KUKA KRL program: EPS_2_26115_SA7004_A_20260219035541.src

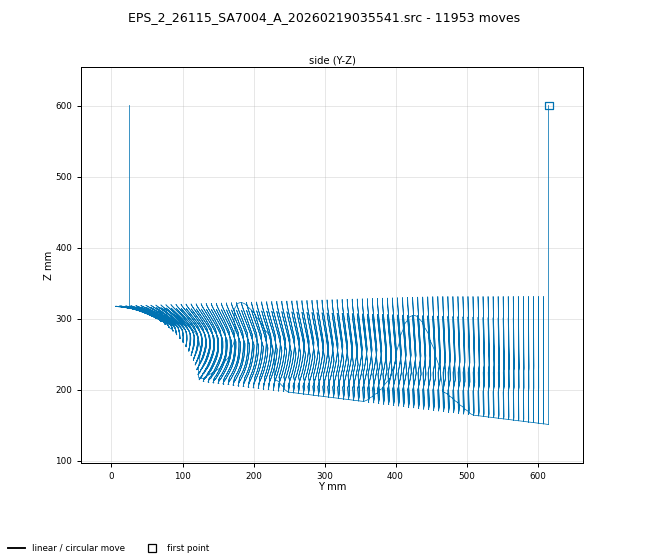
[picture p0: tool path of EPS_2_26115_SA7004_A_20260219035541.src, 11953 of 11955 moves have a stored position in this frame; points joined in program order, loops and branches not executed]
&ACCESS RVP
&REL 4
&COMMENT QRS 19112012
&PARAM EDITMASK = *
DEF PART()
EXT BAS (BAS_COMMAND :IN,REAL :IN )
INT I
BAS (#INITMOV,0 )

;KUKA QRS Post kuka4.cps  Date:22-06-2017 !

File_ID=3058

QRS_PRE_INIT()

;Init var - Until changes are made in qrs_pre_init
Outlet_Square_prg=0
Inlet_1_Square_prg=0
Inlet_2_Square_prg=0
Inlet_3_Square_prg=0
Inlet_4_Square_prg=0
Inlet_5_Square_prg=0

Outlet_1={X 0.000, Y 460.000, Z 230.500, B 0.000, E1 0.000 }
Inlet_1={X 0.000, Y 539.550, Z 200.500, B 0.000, E1 180.000 }
Outlet_1_type=201
Inlet_1_type=201
;QRS#1=Sidecore dimensions
;QRS#2=200-8" PVC SDR 35 Cut Back
;QRS#3=200-8" PVC SDR 35
;QRS#4=
;QRS#5=
;QRS#6=
;QRS#7=
;QRS#8=
;QRS#9=12-08 PSX
;QRS#10=12-08 PSX
;QRS#11=
;QRS#12=
;QRS#13=
;QRS#14=
;QRS#15=
;QRS#16=1220x127x610 2'
;QRS#17=EPS Height
;QRS#18=331
;QRS#19=*
;QRS#20= UPDATED VERSION 22-06-2017
;QRS#21=*
Outlet_Square=0100
Inlet_1_Square=0100
Inlet_2_Square=0
Inlet_3_Square=0
Inlet_4_Square=0
Inlet_5_Square=0
Mill_Square=1
Outlet_Square_Prg=214
Inlet_1_Square_prg=204

QRS_INIT()

$ADVANCE=5

; T1
PTP {E1 173.62,E2 173.62}
PTP {X 0,Y 615.488,A -85,B 0,C 180,E1 173.62,E2 173.62,E3 0,E4 0,E5 0,E6 0}
QRS_SPEED_INIT()
LIN {X 0,Y 615.488,Z 600,A -85,B 0,C 180,E1 173.62,E2 173.62,E3 0,E4 0,E5 0,E6 0} C_VEL
LIN {X 0,Y 615.488,Z 160.871,A -85,B 0,C 180,E1 173.62,E2 173.62} C_VEL
LIN {X 0,Y 615.488,Z 152.699,A -85,B 0,C 180,E1 173.62,E2 173.62} C_VEL
LIN {X 0,Y 615.469,Z 150.699,A -85,B 0,C 180,E1 173.434,E2 173.434} C_VEL
LIN {X 0,Y 615.452,Z 150.696,A -85,B 0,C 180,E1 170.801,E2 170.801} C_VEL
LIN {X 0,Y 615.484,Z 150.7,A -85,B 0,C 180,E1 168.139,E2 168.139} C_VEL
LIN {X 0,Y 615.492,Z 150.686,A -85,B 0,C 180,E1 165.451,E2 165.451} C_VEL
LIN {X 0,Y 615.483,Z 150.699,A -85,B 0,C 180,E1 162.729,E2 162.729} C_VEL
LIN {X 0,Y 615.468,Z 150.694,A -85,B 0,C 180,E1 159.966,E2 159.966} C_VEL
LIN {X 0,Y 615.439,Z 150.7,A -85,B 0,C 180,E1 157.153,E2 157.153} C_VEL
LIN {X 0,Y 615.449,Z 150.697,A -85,B 0,C 180,E1 155.006,E2 155.006} C_VEL
LIN {X 0,Y 615.477,Z 150.698,A -85,B 0,C 180,E1 152.822,E2 152.822} C_VEL
LIN {X 0,Y 615.49,Z 150.688,A -85,B 0,C 180,E1 149.84,E2 149.84} C_VEL
LIN {X 0,Y 615.492,Z 150.699,A -85,B 0,C 180,E1 147.543,E2 147.543} C_VEL
LIN {X 0,Y 615.448,Z 150.698,A -85,B 0,C 180,E1 145.182,E2 145.182} C_VEL
LIN {X 0,Y 615.449,Z 150.7,A -85,B 0,C 180,E1 142.755,E2 142.755} C_VEL
LIN {X 0,Y 615.461,Z 150.694,A -85,B 0,C 180,E1 139.913,E2 139.913} C_VEL
LIN {X 0,Y 615.468,Z 150.695,A -85,B 0,C 180,E1 137.645,E2 137.645} C_VEL
LIN {X 0,Y 615.479,Z 150.691,A -85,B 0,C 180,E1 134.93,E2 134.93} C_VEL
LIN {X 0,Y 615.494,Z 150.7,A -85,B 0,C 180,E1 132.08,E2 132.08} C_VEL
LIN {X 0,Y 615.444,Z 150.699,A -85,B 0,C 180,E1 129.753,E2 129.753} C_VEL
LIN {X 0,Y 615.479,Z 150.704,A -85,B 0,C 180,E1 126.935,E2 126.935} C_VEL
LIN {X 0,Y 615.451,Z 150.699,A -85,B 0,C 180,E1 125.618,E2 125.618} C_VEL
LIN {X 0,Y 615.483,Z 151.858,A -85,B 0,C 180,E1 124.7,E2 124.7} C_VEL
LIN {X 0,Y 615.454,Z 156.021,A -85,B 0,C 180,E1 122.325,E2 122.325} C_VEL
LIN {X 0,Y 615.48,Z 160.511,A -85,B 0,C 180,E1 119.793,E2 119.793} C_VEL
LIN {X 0,Y 615.495,Z 165.513,A -85,B 0,C 180,E1 117.046,E2 117.046} C_VEL
LIN {X 0,Y 615.487,Z 170.773,A -85,B 0,C 180,E1 114.272,E2 114.272} C_VEL
LIN {X 0,Y 615.488,Z 176.264,A -85,B 0,C 180,E1 111.432,E2 111.432} C_VEL
LIN {X 0,Y 615.49,Z 181.84,A -85,B 0,C 180,E1 108.605,E2 108.605} C_VEL
LIN {X 0,Y 615.465,Z 187.255,A -85,B 0,C 180,E1 105.906,E2 105.906} C_VEL
LIN {X 0,Y 615.495,Z 192.741,A -85,B 0,C 180,E1 103.201,E2 103.201} C_VEL
LIN {X 0,Y 615.492,Z 196.091,A -85,B 0,C 180,E1 101.568,E2 101.568} C_VEL
LIN {X 0,Y 615.483,Z 210.748,A -85,B 0,C 180,E1 101.235,E2 101.235} C_VEL
LIN {X 0,Y 615.446,Z 223.1,A -85,B 0,C 180,E1 100.825,E2 100.825} C_VEL
LIN {X 0,Y 615.441,Z 235.207,A -85,B 0,C 180,E1 100.278,E2 100.278} C_VEL
LIN {X 0,Y 615.493,Z 246.579,A -85,B 0,C 180,E1 99.613,E2 99.613} C_VEL
LIN {X 0,Y 615.498,Z 256.825,A -85,B 0,C 180,E1 98.867,E2 98.867} C_VEL
LIN {X 0,Y 615.498,Z 266.036,A -85,B 0,C 180,E1 98.04,E2 98.04} C_VEL
LIN {X 0,Y 615.499,Z 274.893,A -85,B 0,C 180,E1 97.057,E2 97.057} C_VEL
LIN {X 0,Y 615.497,Z 282.125,A -85,B 0,C 180,E1 96.063,E2 96.063} C_VEL
LIN {X 0,Y 615.497,Z 286.959,A -85,B 0,C 180,E1 95.241,E2 95.241} C_VEL
LIN {X 0,Y 615.494,Z 291.659,A -85,B 0,C 180,E1 94.256,E2 94.256} C_VEL
LIN {X 0,Y 615.494,Z 295.255,A -85,B 0,C 180,E1 93.273,E2 93.273} C_VEL
LIN {X 0,Y 615.496,Z 297.115,A -85,B 0,C 180,E1 92.618,E2 92.618} C_VEL
LIN {X 0,Y 615.5,Z 298.533,A -85,B 0,C 180,E1 91.963,E2 91.963} C_VEL
LIN {X 0,Y 615.496,Z 300.142,A -85,B 0,C 180,E1 90.654,E2 90.654} C_VEL
LIN {X 0,Y 615.495,Z 300.384,A -85,B 0,C 180,E1 90,E2 90} C_VEL
LIN {X 0,Y 615.495,Z 300.205,A -85,B 0,C 180,E1 89.346,E2 89.346} C_VEL
LIN {X 0,Y 615.499,Z 298.682,A -85,B 0,C 180,E1 88.037,E2 88.037} C_VEL
LIN {X 0,Y 615.498,Z 297.341,A -85,B 0,C 180,E1 87.382,E2 87.382} C_VEL
LIN {X 0,Y 615.496,Z 294.494,A -85,B 0,C 180,E1 86.399,E2 86.399} C_VEL
LIN {X 0,Y 615.498,Z 290.634,A -85,B 0,C 180,E1 85.415,E2 85.415} C_VEL
LIN {X 0,Y 615.498,Z 285.651,A -85,B 0,C 180,E1 84.43,E2 84.43} C_VEL
LIN {X 0,Y 615.496,Z 279.208,A -85,B 0,C 180,E1 83.418,E2 83.418} C_VEL
LIN {X 0,Y 615.497,Z 271.535,A -85,B 0,C 180,E1 82.454,E2 82.454} C_VEL
LIN {X 0,Y 615.498,Z 261.757,A -85,B 0,C 180,E1 81.463,E2 81.463} C_VEL
LIN {X 0,Y 615.498,Z 251.491,A -85,B 0,C 180,E1 80.636,E2 80.636} C_VEL
LIN {X 0,Y 615.447,Z 239.935,A -85,B 0,C 180,E1 79.888,E2 79.888} C_VEL
LIN {X 0,Y 615.431,Z 228.385,A -85,B 0,C 180,E1 79.305,E2 79.305} C_VEL
LIN {X 0,Y 615.463,Z 216.445,A -85,B 0,C 180,E1 78.848,E2 78.848} C_VEL
LIN {X 0,Y 615.49,Z 204.378,A -85,B 0,C 180,E1 78.515,E2 78.515} C_VEL
LIN {X 0,Y 615.489,Z 196.104,A -85,B 0,C 180,E1 78.348,E2 78.348} C_VEL
LIN {X 0,Y 615.458,Z 191.469,A -85,B 0,C 180,E1 76.08,E2 76.08} C_VEL
LIN {X 0,Y 615.458,Z 186.396,A -85,B 0,C 180,E1 73.579,E2 73.579} C_VEL
LIN {X 0,Y 615.487,Z 180.568,A -85,B 0,C 180,E1 70.662,E2 70.662} C_VEL
LIN {X 0,Y 615.477,Z 175.065,A -85,B 0,C 180,E1 67.863,E2 67.863} C_VEL
LIN {X 0,Y 615.488,Z 169.567,A -85,B 0,C 180,E1 65.008,E2 65.008} C_VEL
LIN {X 0,Y 615.484,Z 164.066,A -85,B 0,C 180,E1 62.085,E2 62.085} C_VEL
LIN {X 0,Y 615.466,Z 160.02,A -85,B 0,C 180,E1 59.839,E2 59.839} C_VEL
LIN {X 0,Y 615.462,Z 155.943,A -85,B 0,C 180,E1 57.541,E2 57.541} C_VEL
LIN {X 0,Y 615.495,Z 151.812,A -85,B 0,C 180,E1 55.185,E2 55.185} C_VEL
LIN {X 0,Y 615.464,Z 150.698,A -85,B 0,C 180,E1 54.383,E2 54.383} C_VEL
LIN {X 0,Y 615.437,Z 150.7,A -85,B 0,C 180,E1 51.928,E2 51.928} C_VEL
LIN {X 0,Y 615.49,Z 150.696,A -85,B 0,C 180,E1 49.394,E2 49.394} C_VEL
LIN {X 0,Y 615.463,Z 150.694,A -85,B 0,C 180,E1 46.753,E2 46.753} C_VEL
LIN {X 0,Y 615.481,Z 150.692,A -85,B 0,C 180,E1 43.997,E2 43.997} C_VEL
LIN {X 0,Y 615.491,Z 150.7,A -85,B 0,C 180,E1 41.095,E2 41.095} C_VEL
LIN {X 0,Y 615.453,Z 150.7,A -85,B 0,C 180,E1 38.907,E2 38.907} C_VEL
LIN {X 0,Y 615.441,Z 150.7,A -85,B 0,C 180,E1 36.428,E2 36.428} C_VEL
LIN {X 0,Y 615.467,Z 150.693,A -85,B 0,C 180,E1 33.531,E2 33.531} C_VEL
LIN {X 0,Y 615.485,Z 150.698,A -85,B 0,C 180,E1 30.92,E2 30.92} C_VEL
LIN {X 0,Y 615.479,Z 150.691,A -85,B 0,C 180,E1 28.449,E2 28.449} C_VEL
LIN {X 0,Y 615.493,Z 150.7,A -85,B 0,C 180,E1 25.57,E2 25.57} C_VEL
LIN {X 0,Y 615.458,Z 150.7,A -85,B 0,C 180,E1 23.558,E2 23.558} C_VEL
LIN {X 0,Y 615.432,Z 150.7,A -85,B 0,C 180,E1 21.434,E2 21.434} C_VEL
LIN {X 0,Y 615.494,Z 150.696,A -85,B 0,C 180,E1 18.606,E2 18.606} C_VEL
LIN {X 0,Y 615.472,Z 150.693,A -85,B 0,C 180,E1 15.906,E2 15.906} C_VEL
LIN {X 0,Y 615.475,Z 150.694,A -85,B 0,C 180,E1 13.202,E2 13.202} C_VEL
LIN {X 0,Y 615.492,Z 150.693,A -85,B 0,C 180,E1 10.527,E2 10.527} C_VEL
LIN {X 0,Y 615.437,Z 150.7,A -85,B 0,C 180,E1 7.876,E2 7.876} C_VEL
LIN {X 0,Y 615.474,Z 150.701,A -85,B 0,C 180,E1 5.241,E2 5.241} C_VEL
LIN {X 0,Y 615.474,Z 150.691,A -85,B 0,C 180,E1 2.618,E2 2.618} C_VEL
LIN {X 0,Y 615.487,Z 150.701,A -85,B 0,C 180,E1 0,E2 0} C_VEL
LIN {X 0,Y 615.478,Z 150.69,A -85,B 0,C 180,E1 -2.618,E2 -2.618} C_VEL
LIN {X 0,Y 615.489,Z 150.701,A -85,B 0,C 180,E1 -5.241,E2 -5.241} C_VEL
LIN {X 0,Y 615.433,Z 150.7,A -85,B 0,C 180,E1 -7.876,E2 -7.876} C_VEL
LIN {X 0,Y 615.494,Z 150.695,A -85,B 0,C 180,E1 -10.527,E2 -10.527} C_VEL
LIN {X 0,Y 615.468,Z 150.694,A -85,B 0,C 180,E1 -13.202,E2 -13.202} C_VEL
LIN {X 0,Y 615.478,Z 150.693,A -85,B 0,C 180,E1 -15.905,E2 -15.905} C_VEL
LIN {X 0,Y 615.494,Z 150.694,A -85,B 0,C 180,E1 -18.646,E2 -18.646} C_VEL
LIN {X 0,Y 615.436,Z 150.699,A -85,B 0,C 180,E1 -21.434,E2 -21.434} C_VEL
LIN {X 0,Y 615.484,Z 150.696,A -85,B 0,C 180,E1 -24.272,E2 -24.272} C_VEL
LIN {X 0,Y 615.471,Z 150.692,A -85,B 0,C 180,E1 -26.445,E2 -26.445} C_VEL
LIN {X 0,Y 615.472,Z 150.694,A -85,B 0,C 180,E1 -28.659,E2 -28.659} C_VEL
LIN {X 0,Y 615.481,Z 150.698,A -85,B 0,C 180,E1 -31.085,E2 -31.085} C_VEL
LIN {X 0,Y 615.47,Z 150.691,A -85,B 0,C 180,E1 -33.532,E2 -33.532} C_VEL
LIN {X 0,Y 615.45,Z 150.7,A -85,B 0,C 180,E1 -36.427,E2 -36.427} C_VEL
LIN {X 0,Y 615.454,Z 150.7,A -85,B 0,C 180,E1 -39.058,E2 -39.058} C_VEL
LIN {X 0,Y 615.494,Z 150.692,A -85,B 0,C 180,E1 -41.473,E2 -41.473} C_VEL
LIN {X 0,Y 615.477,Z 150.694,A -85,B 0,C 180,E1 -44.151,E2 -44.151} C_VEL
LIN {X 0,Y 615.471,Z 150.692,A -85,B 0,C 180,E1 -46.954,E2 -46.954} C_VEL
LIN {X 0,Y 615.489,Z 150.693,A -85,B 0,C 180,E1 -49.394,E2 -49.394} C_VEL
LIN {X 0,Y 615.439,Z 150.7,A -85,B 0,C 180,E1 -51.994,E2 -51.994} C_VEL
LIN {X 0,Y 615.468,Z 150.791,A -85,B 0,C 180,E1 -54.584,E2 -54.584} C_VEL
LIN {X 0,Y 615.484,Z 158.007,A -85,B 0,C 180,E1 -57.154,E2 -57.154} C_VEL
LIN {X 0,Y 615.463,Z 165.783,A -85,B 0,C 180,E1 -59.839,E2 -59.839} C_VEL
LIN {X 0,Y 615.486,Z 173.542,A -85,B 0,C 180,E1 -62.454,E2 -62.454} C_VEL
LIN {X 0,Y 615.487,Z 181.309,A -85,B 0,C 180,E1 -65.008,E2 -65.008} C_VEL
LIN {X 0,Y 615.481,Z 190.171,A -85,B 0,C 180,E1 -67.863,E2 -67.863} C_VEL
LIN {X 0,Y 615.488,Z 199.041,A -85,B 0,C 180,E1 -70.662,E2 -70.662} C_VEL
LIN {X 0,Y 615.471,Z 207.89,A -85,B 0,C 180,E1 -73.413,E2 -73.413} C_VEL
LIN {X 0,Y 615.46,Z 216.602,A -85,B 0,C 180,E1 -76.079,E2 -76.079} C_VEL
LIN {X 0,Y 615.491,Z 224.137,A -85,B 0,C 180,E1 -78.369,E2 -78.369} C_VEL
LIN {X 0,Y 615.497,Z 237.817,A -85,B 0,C 180,E1 -78.64,E2 -78.64} C_VEL
LIN {X 0,Y 615.449,Z 251.023,A -85,B 0,C 180,E1 -79.053,E2 -79.053} C_VEL
LIN {X 0,Y 615.433,Z 262.772,A -85,B 0,C 180,E1 -79.555,E2 -79.555} C_VEL
LIN {X 0,Y 615.474,Z 273.388,A -85,B 0,C 180,E1 -80.137,E2 -80.137} C_VEL
LIN {X 0,Y 615.498,Z 284.23,A -85,B 0,C 180,E1 -80.884,E2 -80.884} C_VEL
LIN {X 0,Y 615.497,Z 294.81,A -85,B 0,C 180,E1 -81.794,E2 -81.794} C_VEL
LIN {X 0,Y 615.498,Z 302.605,A -85,B 0,C 180,E1 -82.619,E2 -82.619} C_VEL
LIN {X 0,Y 615.496,Z 310.202,A -85,B 0,C 180,E1 -83.608,E2 -83.608} C_VEL
LIN {X 0,Y 615.498,Z 317.204,A -85,B 0,C 180,E1 -84.759,E2 -84.759} C_VEL
LIN {X 0,Y 615.493,Z 321.851,A -85,B 0,C 180,E1 -85.743,E2 -85.743} C_VEL
LIN {X 0,Y 615.494,Z 325.398,A -85,B 0,C 180,E1 -86.727,E2 -86.727} C_VEL
LIN {X 0,Y 615.497,Z 327.233,A -85,B 0,C 180,E1 -87.382,E2 -87.382} C_VEL
LIN {X 0,Y 615.5,Z 328.607,A -85,B 0,C 180,E1 -88.037,E2 -88.037} C_VEL
LIN {X 0,Y 615.496,Z 330.173,A -85,B 0,C 180,E1 -89.346,E2 -89.346} C_VEL
LIN {X 0,Y 615.494,Z 330.389,A -85,B 0,C 180,E1 -90,E2 -90} C_VEL
LIN {X 0,Y 615.495,Z 329.58,A -85,B 0,C 180,E1 -91.308,E2 -91.308} C_VEL
LIN {X 0,Y 615.5,Z 328.608,A -85,B 0,C 180,E1 -91.963,E2 -91.963} C_VEL
LIN {X 0,Y 615.497,Z 327.233,A -85,B 0,C 180,E1 -92.618,E2 -92.618} C_VEL
LIN {X 0,Y 615.496,Z 324.35,A -85,B 0,C 180,E1 -93.6,E2 -93.6} C_VEL
LIN {X 0,Y 615.498,Z 320.442,A -85,B 0,C 180,E1 -94.584,E2 -94.584} C_VEL
LIN {X 0,Y 615.499,Z 315.406,A -85,B 0,C 180,E1 -95.569,E2 -95.569} C_VEL
LIN {X 0,Y 615.497,Z 308.869,A -85,B 0,C 180,E1 -96.583,E2 -96.583} C_VEL
LIN {X 0,Y 615.498,Z 301.135,A -85,B 0,C 180,E1 -97.545,E2 -97.545} C_VEL
LIN {X 0,Y 615.498,Z 293.047,A -85,B 0,C 180,E1 -98.371,E2 -98.371} C_VEL
LIN {X 0,Y 615.499,Z 283.17,A -85,B 0,C 180,E1 -99.198,E2 -99.198} C_VEL
LIN {X 0,Y 615.464,Z 271.989,A -85,B 0,C 180,E1 -99.945,E2 -99.945} C_VEL
LIN {X 0,Y 615.432,Z 261.036,A -85,B 0,C 180,E1 -100.528,E2 -100.528} C_VEL
LIN {X 0,Y 615.456,Z 248.815,A -85,B 0,C 180,E1 -101.029,E2 -101.029} C_VEL
LIN {X 0,Y 615.498,Z 236.072,A -85,B 0,C 180,E1 -101.401,E2 -101.401} C_VEL
LIN {X 0,Y 615.491,Z 224.138,A -85,B 0,C 180,E1 -101.631,E2 -101.631} C_VEL
LIN {X 0,Y 615.448,Z 215.568,A -85,B 0,C 180,E1 -104.235,E2 -104.235} C_VEL
LIN {X 0,Y 615.492,Z 206.782,A -85,B 0,C 180,E1 -106.928,E2 -106.928} C_VEL
LIN {X 0,Y 615.474,Z 197.931,A -85,B 0,C 180,E1 -109.685,E2 -109.685} C_VEL
LIN {X 0,Y 615.49,Z 189.513,A -85,B 0,C 180,E1 -112.346,E2 -112.346} C_VEL
LIN {X 0,Y 615.487,Z 181.31,A -85,B 0,C 180,E1 -114.991,E2 -114.991} C_VEL
LIN {X 0,Y 615.484,Z 172.435,A -85,B 0,C 180,E1 -117.915,E2 -117.915} C_VEL
LIN {X 0,Y 615.466,Z 164.672,A -85,B 0,C 180,E1 -120.54,E2 -120.54} C_VEL
LIN {X 0,Y 615.495,Z 156.897,A -85,B 0,C 180,E1 -123.235,E2 -123.235} C_VEL
LIN {X 0,Y 615.458,Z 150.699,A -85,B 0,C 180,E1 -125.517,E2 -125.517} C_VEL
LIN {X 0,Y 615.443,Z 150.7,A -85,B 0,C 180,E1 -128.071,E2 -128.071} C_VEL
LIN {X 0,Y 615.489,Z 150.693,A -85,B 0,C 180,E1 -130.606,E2 -130.606} C_VEL
LIN {X 0,Y 615.47,Z 150.694,A -85,B 0,C 180,E1 -133.246,E2 -133.246} C_VEL
LIN {X 0,Y 615.476,Z 150.692,A -85,B 0,C 180,E1 -136.003,E2 -136.003} C_VEL
LIN {X 0,Y 615.484,Z 150.702,A -85,B 0,C 180,E1 -138.905,E2 -138.905} C_VEL
LIN {X 0,Y 615.444,Z 150.7,A -85,B 0,C 180,E1 -141.092,E2 -141.092} C_VEL
LIN {X 0,Y 615.492,Z 150.697,A -85,B 0,C 180,E1 -144.165,E2 -144.165} C_VEL
LIN {X 0,Y 615.461,Z 150.694,A -85,B 0,C 180,E1 -146.762,E2 -146.762} C_VEL
LIN {X 0,Y 615.494,Z 150.699,A -85,B 0,C 180,E1 -149.081,E2 -149.081} C_VEL
LIN {X 0,Y 615.475,Z 150.691,A -85,B 0,C 180,E1 -151.551,E2 -151.551} C_VEL
LIN {X 0,Y 615.48,Z 150.7,A -85,B 0,C 180,E1 -154.432,E2 -154.432} C_VEL
LIN {X 0,Y 615.448,Z 150.7,A -85,B 0,C 180,E1 -156.442,E2 -156.442} C_VEL
LIN {X 0,Y 615.434,Z 150.699,A -85,B 0,C 180,E1 -158.566,E2 -158.566} C_VEL
LIN {X 0,Y 615.494,Z 150.694,A -85,B 0,C 180,E1 -161.392,E2 -161.392} C_VEL
LIN {X 0,Y 615.474,Z 150.694,A -85,B 0,C 180,E1 -164.094,E2 -164.094} C_VEL
LIN {X 0,Y 615.47,Z 150.694,A -85,B 0,C 180,E1 -166.798,E2 -166.798} C_VEL
LIN {X 0,Y 615.493,Z 150.694,A -85,B 0,C 180,E1 -169.473,E2 -169.473} C_VEL
LIN {X 0,Y 615.434,Z 150.7,A -85,B 0,C 180,E1 -172.124,E2 -172.124} C_VEL
LIN {X 0,Y 615.484,Z 150.701,A -85,B 0,C 180,E1 -174.759,E2 -174.759} C_VEL
LIN {X 0,Y 615.476,Z 150.69,A -85,B 0,C 180,E1 -177.382,E2 -177.382} C_VEL
LIN {X 0,Y 615.487,Z 150.703,A -85,B 0,C 180,E1 -180,E2 -180} C_VEL
LIN {X 0,Y 615.476,Z 150.69,A -85,B 0,C 180,E1 -182.618,E2 -182.618} C_VEL
LIN {X 0,Y 615.48,Z 150.701,A -85,B 0,C 180,E1 -185.241,E2 -185.241} C_VEL
LIN {X 0,Y 615.469,Z 150.699,A -85,B 0,C 180,E1 -186.566,E2 -186.566} C_VEL
LIN {X 0,Y 614.782,Z 150.847,A -85,B 0,C 180,E1 -187.112,E2 -187.112} C_VEL
LIN {X 0,Y 611.94,Z 151.257,A -85,B 0,C 180,E1 -187.998,E2 -187.998} C_VEL
LIN {X 0,Y 609.549,Z 151.565,A -85,B 0,C 180,E1 -188.71,E2 -188.71} C_VEL
LIN {X 0,Y 608.518,Z 151.683,A -85,B 0,C 180,E1 -189.26,E2 -189.26} C_VEL
LIN {X 0,Y 608.431,Z 151.693,A -85,B 0,C 180,E1 -189.446,E2 -189.446} C_VEL
LIN {X 0,Y 608.462,Z 151.697,A -85,B 0,C 180,E1 -192,E2 -192} C_VEL
LIN {X 0,Y 608.479,Z 151.687,A -85,B 0,C 180,E1 -194.721,E2 -194.721} C_VEL
LIN {X 0,Y 608.445,Z 151.694,A -85,B 0,C 180,E1 -197.477,E2 -197.477} C_VEL
LIN {X 0,Y 608.427,Z 151.693,A -85,B 0,C 180,E1 -199.572,E2 -199.572} C_VEL
LIN {X 0,Y 608.434,Z 151.693,A -85,B 0,C 180,E1 -201.693,E2 -201.693} C_VEL
LIN {X 0,Y 608.439,Z 151.692,A -85,B 0,C 180,E1 -204.572,E2 -204.572} C_VEL
LIN {X 0,Y 608.471,Z 151.693,A -85,B 0,C 180,E1 -207.207,E2 -207.207} C_VEL
LIN {X 0,Y 608.469,Z 151.688,A -85,B 0,C 180,E1 -209.972,E2 -209.972} C_VEL
LIN {X 0,Y 608.447,Z 151.694,A -85,B 0,C 180,E1 -212.88,E2 -212.88} C_VEL
LIN {X 0,Y 608.423,Z 151.694,A -85,B 0,C 180,E1 -215.279,E2 -215.279} C_VEL
LIN {X 0,Y 608.444,Z 151.692,A -85,B 0,C 180,E1 -218.238,E2 -218.238} C_VEL
LIN {X 0,Y 608.466,Z 151.693,A -85,B 0,C 180,E1 -221.343,E2 -221.343} C_VEL
LIN {X 0,Y 608.449,Z 151.695,A -85,B 0,C 180,E1 -224.264,E2 -224.264} C_VEL
LIN {X 0,Y 608.439,Z 151.692,A -85,B 0,C 180,E1 -227.039,E2 -227.039} C_VEL
LIN {X 0,Y 608.453,Z 151.698,A -85,B 0,C 180,E1 -229.697,E2 -229.697} C_VEL
LIN {X 0,Y 608.459,Z 151.693,A -85,B 0,C 180,E1 -232.843,E2 -232.843} C_VEL
LIN {X 0,Y 608.4,Z 151.86,A -85,B 0,C 180,E1 -234.72,E2 -234.72} C_VEL
LIN {X 0,Y 608.44,Z 156.641,A -85,B 0,C 180,E1 -237.481,E2 -237.481} C_VEL
LIN {X 0,Y 608.465,Z 161.459,A -85,B 0,C 180,E1 -240.221,E2 -240.221} C_VEL
LIN {X 0,Y 608.426,Z 166.89,A -85,B 0,C 180,E1 -243.225,E2 -243.225} C_VEL
LIN {X 0,Y 608.458,Z 171.842,A -85,B 0,C 180,E1 -245.852,E2 -245.852} C_VEL
LIN {X 0,Y 608.445,Z 176.566,A -85,B 0,C 180,E1 -248.308,E2 -248.308} C_VEL
LIN {X 0,Y 608.429,Z 182.425,A -85,B 0,C 180,E1 -251.297,E2 -251.297} C_VEL
LIN {X 0,Y 608.425,Z 187.625,A -85,B 0,C 180,E1 -253.905,E2 -253.905} C_VEL
LIN {X 0,Y 608.43,Z 193.155,A -85,B 0,C 180,E1 -256.643,E2 -256.643} C_VEL
LIN {X 0,Y 608.443,Z 196.525,A -85,B 0,C 180,E1 -258.296,E2 -258.296} C_VEL
LIN {X 0,Y 608.53,Z 212.4,A -85,B 0,C 180,E1 -258.677,E2 -258.677} C_VEL
LIN {X 0,Y 608.478,Z 224.8,A -85,B 0,C 180,E1 -259.113,E2 -259.113} C_VEL
LIN {X 0,Y 608.444,Z 236.939,A -85,B 0,C 180,E1 -259.687,E2 -259.687} C_VEL
LIN {X 0,Y 608.492,Z 248.07,A -85,B 0,C 180,E1 -260.359,E2 -260.359} C_VEL
LIN {X 0,Y 608.474,Z 257.086,A -85,B 0,C 180,E1 -261.03,E2 -261.03} C_VEL
LIN {X 0,Y 608.464,Z 266.352,A -85,B 0,C 180,E1 -261.866,E2 -261.866} C_VEL
LIN {X 0,Y 608.466,Z 275.325,A -85,B 0,C 180,E1 -262.868,E2 -262.868} C_VEL
LIN {X 0,Y 608.444,Z 282.557,A -85,B 0,C 180,E1 -263.867,E2 -263.867} C_VEL
LIN {X 0,Y 608.462,Z 287.435,A -85,B 0,C 180,E1 -264.698,E2 -264.698} C_VEL
LIN {X 0,Y 608.439,Z 292.179,A -85,B 0,C 180,E1 -265.694,E2 -265.694} C_VEL
LIN {X 0,Y 608.425,Z 295.813,A -85,B 0,C 180,E1 -266.689,E2 -266.689} C_VEL
LIN {X 0,Y 608.425,Z 297.691,A -85,B 0,C 180,E1 -267.352,E2 -267.352} C_VEL
LIN {X 0,Y 608.445,Z 299.127,A -85,B 0,C 180,E1 -268.014,E2 -268.014} C_VEL
LIN {X 0,Y 608.439,Z 300.752,A -85,B 0,C 180,E1 -269.338,E2 -269.338} C_VEL
LIN {X 0,Y 608.435,Z 300.995,A -85,B 0,C 180,E1 -270,E2 -270} C_VEL
LIN {X 0,Y 608.438,Z 300.815,A -85,B 0,C 180,E1 -270.662,E2 -270.662} C_VEL
LIN {X 0,Y 608.444,Z 299.276,A -85,B 0,C 180,E1 -271.986,E2 -271.986} C_VEL
LIN {X 0,Y 608.426,Z 297.918,A -85,B 0,C 180,E1 -272.648,E2 -272.648} C_VEL
LIN {X 0,Y 608.449,Z 295.041,A -85,B 0,C 180,E1 -273.643,E2 -273.643} C_VEL
LIN {X 0,Y 608.433,Z 291.142,A -85,B 0,C 180,E1 -274.638,E2 -274.638} C_VEL
LIN {X 0,Y 608.45,Z 286.111,A -85,B 0,C 180,E1 -275.635,E2 -275.635} C_VEL
LIN {X 0,Y 608.441,Z 279.794,A -85,B 0,C 180,E1 -276.633,E2 -276.633} C_VEL
LIN {X 0,Y 608.475,Z 271.877,A -85,B 0,C 180,E1 -277.633,E2 -277.633} C_VEL
LIN {X 0,Y 608.472,Z 262.035,A -85,B 0,C 180,E1 -278.636,E2 -278.636} C_VEL
LIN {X 0,Y 608.48,Z 251.712,A -85,B 0,C 180,E1 -279.473,E2 -279.473} C_VEL
LIN {X 0,Y 608.442,Z 240.098,A -85,B 0,C 180,E1 -280.23,E2 -280.23} C_VEL
LIN {X 0,Y 608.461,Z 228.507,A -85,B 0,C 180,E1 -280.819,E2 -280.819} C_VEL
LIN {X 0,Y 608.493,Z 216.426,A -85,B 0,C 180,E1 -281.285,E2 -281.285} C_VEL
LIN {X 0,Y 608.531,Z 203.554,A -85,B 0,C 180,E1 -281.639,E2 -281.639} C_VEL
LIN {X 0,Y 608.432,Z 196.535,A -85,B 0,C 180,E1 -281.789,E2 -281.789} C_VEL
LIN {X 0,Y 608.402,Z 191.954,A -85,B 0,C 180,E1 -284.039,E2 -284.039} C_VEL
LIN {X 0,Y 608.409,Z 186.422,A -85,B 0,C 180,E1 -286.785,E2 -286.785} C_VEL
LIN {X 0,Y 608.427,Z 180.89,A -85,B 0,C 180,E1 -289.572,E2 -289.572} C_VEL
LIN {X 0,Y 608.436,Z 175.357,A -85,B 0,C 180,E1 -292.407,E2 -292.407} C_VEL
LIN {X 0,Y 608.425,Z 171.207,A -85,B 0,C 180,E1 -294.572,E2 -294.572} C_VEL
LIN {X 0,Y 608.443,Z 166.265,A -85,B 0,C 180,E1 -297.2,E2 -297.2} C_VEL
LIN {X 0,Y 608.446,Z 161.295,A -85,B 0,C 180,E1 -299.968,E2 -299.968} C_VEL
LIN {X 0,Y 608.453,Z 156.167,A -85,B 0,C 180,E1 -302.88,E2 -302.88} C_VEL
LIN {X 0,Y 608.435,Z 152.013,A -85,B 0,C 180,E1 -305.278,E2 -305.278} C_VEL
LIN {X 0,Y 608.457,Z 151.697,A -85,B 0,C 180,E1 -306.915,E2 -306.915} C_VEL
LIN {X 0,Y 608.412,Z 151.695,A -85,B 0,C 180,E1 -309.444,E2 -309.444} C_VEL
LIN {X 0,Y 608.466,Z 151.693,A -85,B 0,C 180,E1 -312.334,E2 -312.334} C_VEL
LIN {X 0,Y 608.448,Z 151.691,A -85,B 0,C 180,E1 -314.797,E2 -314.797} C_VEL
LIN {X 0,Y 608.451,Z 151.695,A -85,B 0,C 180,E1 -317.04,E2 -317.04} C_VEL
LIN {X 0,Y 608.454,Z 151.69,A -85,B 0,C 180,E1 -319.697,E2 -319.697} C_VEL
LIN {X 0,Y 608.45,Z 151.696,A -85,B 0,C 180,E1 -322.252,E2 -322.252} C_VEL
LIN {X 0,Y 608.41,Z 151.696,A -85,B 0,C 180,E1 -325.1,E2 -325.1} C_VEL
LIN {X 0,Y 608.47,Z 151.691,A -85,B 0,C 180,E1 -327.906,E2 -327.906} C_VEL
LIN {X 0,Y 608.47,Z 151.688,A -85,B 0,C 180,E1 -330.22,E2 -330.22} C_VEL
LIN {X 0,Y 608.475,Z 151.693,A -85,B 0,C 180,E1 -332.793,E2 -332.793} C_VEL
LIN {X 0,Y 608.441,Z 151.692,A -85,B 0,C 180,E1 -335.428,E2 -335.428} C_VEL
LIN {X 0,Y 608.437,Z 151.693,A -85,B 0,C 180,E1 -338.307,E2 -338.307} C_VEL
LIN {X 0,Y 608.451,Z 151.697,A -85,B 0,C 180,E1 -341.13,E2 -341.13} C_VEL
LIN {X 0,Y 608.454,Z 151.69,A -85,B 0,C 180,E1 -343.906,E2 -343.906} C_VEL
LIN {X 0,Y 608.455,Z 151.694,A -85,B 0,C 180,E1 -346.643,E2 -346.643} C_VEL
LIN {X 0,Y 608.465,Z 151.69,A -85,B 0,C 180,E1 -349.35,E2 -349.35} C_VEL
LIN {X 0,Y 608.411,Z 151.696,A -85,B 0,C 180,E1 -352.032,E2 -352.032} C_VEL
LIN {X 0,Y 608.45,Z 151.695,A -85,B 0,C 180,E1 -354.698,E2 -354.698} C_VEL
LIN {X 0,Y 608.467,Z 151.688,A -85,B 0,C 180,E1 -357.352,E2 -357.352} C_VEL
LIN {X 0,Y 608.477,Z 151.694,A -85,B 0,C 180,E1 -360,E2 -360} C_VEL
LIN {X 0,Y 608.47,Z 151.688,A -85,B 0,C 180,E1 -362.648,E2 -362.648} C_VEL
LIN {X 0,Y 608.463,Z 151.695,A -85,B 0,C 180,E1 -365.302,E2 -365.302} C_VEL
LIN {X 0,Y 608.406,Z 151.696,A -85,B 0,C 180,E1 -367.968,E2 -367.968} C_VEL
LIN {X 0,Y 608.465,Z 151.692,A -85,B 0,C 180,E1 -370.65,E2 -370.65} C_VEL
LIN {X 0,Y 608.452,Z 151.693,A -85,B 0,C 180,E1 -373.357,E2 -373.357} C_VEL
LIN {X 0,Y 608.457,Z 151.69,A -85,B 0,C 180,E1 -376.094,E2 -376.094} C_VEL
LIN {X 0,Y 608.454,Z 151.698,A -85,B 0,C 180,E1 -378.87,E2 -378.87} C_VEL
LIN {X 0,Y 608.438,Z 151.693,A -85,B 0,C 180,E1 -381.693,E2 -381.693} C_VEL
LIN {X 0,Y 608.437,Z 151.693,A -85,B 0,C 180,E1 -384.572,E2 -384.572} C_VEL
LIN {X 0,Y 608.468,Z 151.692,A -85,B 0,C 180,E1 -387.205,E2 -387.205} C_VEL
LIN {X 0,Y 608.469,Z 151.688,A -85,B 0,C 180,E1 -389.972,E2 -389.972} C_VEL
LIN {X 0,Y 608.448,Z 151.694,A -85,B 0,C 180,E1 -392.88,E2 -392.88} C_VEL
LIN {X 0,Y 608.425,Z 151.694,A -85,B 0,C 180,E1 -395.279,E2 -395.279} C_VEL
LIN {X 0,Y 608.445,Z 151.699,A -85,B 0,C 180,E1 -397.748,E2 -397.748} C_VEL
LIN {X 0,Y 608.433,Z 151.692,A -85,B 0,C 180,E1 -400.327,E2 -400.327} C_VEL
LIN {X 0,Y 608.454,Z 151.696,A -85,B 0,C 180,E1 -402.96,E2 -402.96} C_VEL
LIN {X 0,Y 608.453,Z 151.691,A -85,B 0,C 180,E1 -405.737,E2 -405.737} C_VEL
LIN {X 0,Y 608.439,Z 151.692,A -85,B 0,C 180,E1 -408.661,E2 -408.661} C_VEL
LIN {X 0,Y 608.417,Z 151.703,A -85,B 0,C 180,E1 -411.408,E2 -411.408} C_VEL
LIN {X 0,Y 608.432,Z 151.694,A -85,B 0,C 180,E1 -413.957,E2 -413.957} C_VEL
LIN {X 0,Y 608.443,Z 151.795,A -85,B 0,C 180,E1 -414.469,E2 -414.469} C_VEL
LIN {X 0,Y 608.494,Z 159.169,A -85,B 0,C 180,E1 -417.123,E2 -417.123} C_VEL
LIN {X 0,Y 608.48,Z 167.507,A -85,B 0,C 180,E1 -420.027,E2 -420.027} C_VEL
LIN {X 0,Y 608.485,Z 175.673,A -85,B 0,C 180,E1 -422.792,E2 -422.792} C_VEL
LIN {X 0,Y 608.457,Z 183.656,A -85,B 0,C 180,E1 -425.429,E2 -425.429} C_VEL
LIN {X 0,Y 608.442,Z 191.447,A -85,B 0,C 180,E1 -427.951,E2 -427.951} C_VEL
LIN {X 0,Y 608.453,Z 199.239,A -85,B 0,C 180,E1 -430.429,E2 -430.429} C_VEL
LIN {X 0,Y 608.45,Z 208.143,A -85,B 0,C 180,E1 -433.216,E2 -433.216} C_VEL
LIN {X 0,Y 608.424,Z 217.048,A -85,B 0,C 180,E1 -435.961,E2 -435.961} C_VEL
LIN {X 0,Y 608.428,Z 224.491,A -85,B 0,C 180,E1 -438.232,E2 -438.232} C_VEL
LIN {X 0,Y 608.544,Z 238.692,A -85,B 0,C 180,E1 -438.53,E2 -438.53} C_VEL
LIN {X 0,Y 608.492,Z 251.84,A -85,B 0,C 180,E1 -438.952,E2 -438.952} C_VEL
LIN {X 0,Y 608.463,Z 262.918,A -85,B 0,C 180,E1 -439.434,E2 -439.434} C_VEL
LIN {X 0,Y 608.463,Z 273.576,A -85,B 0,C 180,E1 -440.023,E2 -440.023} C_VEL
LIN {X 0,Y 608.483,Z 284.472,A -85,B 0,C 180,E1 -440.778,E2 -440.778} C_VEL
LIN {X 0,Y 608.475,Z 295.11,A -85,B 0,C 180,E1 -441.699,E2 -441.699} C_VEL
LIN {X 0,Y 608.471,Z 302.959,A -85,B 0,C 180,E1 -442.534,E2 -442.534} C_VEL
LIN {X 0,Y 608.461,Z 310.286,A -85,B 0,C 180,E1 -443.484,E2 -443.484} C_VEL
LIN {X 0,Y 608.45,Z 315.865,A -85,B 0,C 180,E1 -444.365,E2 -444.365} C_VEL
LIN {X 0,Y 608.432,Z 320.949,A -85,B 0,C 180,E1 -445.362,E2 -445.362} C_VEL
LIN {X 0,Y 608.449,Z 324.896,A -85,B 0,C 180,E1 -446.357,E2 -446.357} C_VEL
LIN {X 0,Y 608.425,Z 327.809,A -85,B 0,C 180,E1 -447.352,E2 -447.352} C_VEL
LIN {X 0,Y 608.444,Z 329.201,A -85,B 0,C 180,E1 -448.014,E2 -448.014} C_VEL
LIN {X 0,Y 608.438,Z 330.783,A -85,B 0,C 180,E1 -449.338,E2 -449.338} C_VEL
LIN {X 0,Y 608.434,Z 331,A -85,B 0,C 180,E1 -450,E2 -450} C_VEL
LIN {X 0,Y 608.448,Z 330.184,A -85,B 0,C 180,E1 -451.324,E2 -451.324} C_VEL
LIN {X 0,Y 608.444,Z 329.202,A -85,B 0,C 180,E1 -451.986,E2 -451.986} C_VEL
LIN {X 0,Y 608.425,Z 327.81,A -85,B 0,C 180,E1 -452.648,E2 -452.648} C_VEL
LIN {X 0,Y 608.449,Z 324.897,A -85,B 0,C 180,E1 -453.642,E2 -453.642} C_VEL
LIN {X 0,Y 608.432,Z 320.951,A -85,B 0,C 180,E1 -454.638,E2 -454.638} C_VEL
LIN {X 0,Y 608.438,Z 314.878,A -85,B 0,C 180,E1 -455.801,E2 -455.801} C_VEL
LIN {X 0,Y 608.462,Z 308.236,A -85,B 0,C 180,E1 -456.799,E2 -456.799} C_VEL
LIN {X 0,Y 608.456,Z 299.991,A -85,B 0,C 180,E1 -457.8,E2 -457.8} C_VEL
LIN {X 0,Y 608.472,Z 291.538,A -85,B 0,C 180,E1 -458.636,E2 -458.636} C_VEL
LIN {X 0,Y 608.48,Z 281.093,A -85,B 0,C 180,E1 -459.473,E2 -459.473} C_VEL
LIN {X 0,Y 608.459,Z 270.758,A -85,B 0,C 180,E1 -460.145,E2 -460.145} C_VEL
LIN {X 0,Y 608.459,Z 259.89,A -85,B 0,C 180,E1 -460.712,E2 -460.712} C_VEL
LIN {X 0,Y 608.491,Z 248.116,A -85,B 0,C 180,E1 -461.185,E2 -461.185} C_VEL
LIN {X 0,Y 608.547,Z 235.276,A -85,B 0,C 180,E1 -461.554,E2 -461.554} C_VEL
LIN {X 0,Y 608.428,Z 224.492,A -85,B 0,C 180,E1 -461.768,E2 -461.768} C_VEL
LIN {X 0,Y 608.395,Z 215.936,A -85,B 0,C 180,E1 -464.38,E2 -464.38} C_VEL
LIN {X 0,Y 608.449,Z 208.144,A -85,B 0,C 180,E1 -466.784,E2 -466.784} C_VEL
LIN {X 0,Y 608.452,Z 199.24,A -85,B 0,C 180,E1 -469.57,E2 -469.57} C_VEL
LIN {X 0,Y 608.479,Z 190.336,A -85,B 0,C 180,E1 -472.405,E2 -472.405} C_VEL
LIN {X 0,Y 608.471,Z 182.544,A -85,B 0,C 180,E1 -474.934,E2 -474.934} C_VEL
LIN {X 0,Y 608.467,Z 173.64,A -85,B 0,C 180,E1 -477.891,E2 -477.891} C_VEL
LIN {X 0,Y 608.465,Z 165.848,A -85,B 0,C 180,E1 -480.545,E2 -480.545} C_VEL
LIN {X 0,Y 608.519,Z 158.057,A -85,B 0,C 180,E1 -483.27,E2 -483.27} C_VEL
LIN {X 0,Y 608.432,Z 151.696,A -85,B 0,C 180,E1 -485.583,E2 -485.583} C_VEL
LIN {X 0,Y 608.435,Z 151.695,A -85,B 0,C 180,E1 -488.236,E2 -488.236} C_VEL
LIN {X 0,Y 608.43,Z 151.693,A -85,B 0,C 180,E1 -491.178,E2 -491.178} C_VEL
LIN {X 0,Y 608.469,Z 151.694,A -85,B 0,C 180,E1 -493.869,E2 -493.869} C_VEL
LIN {X 0,Y 608.476,Z 151.689,A -85,B 0,C 180,E1 -496.69,E2 -496.69} C_VEL
LIN {X 0,Y 608.455,Z 151.697,A -85,B 0,C 180,E1 -498.823,E2 -498.823} C_VEL
LIN {X 0,Y 608.443,Z 151.692,A -85,B 0,C 180,E1 -501.762,E2 -501.762} C_VEL
LIN {X 0,Y 608.426,Z 151.694,A -85,B 0,C 180,E1 -504.721,E2 -504.721} C_VEL
LIN {X 0,Y 608.465,Z 151.696,A -85,B 0,C 180,E1 -507.476,E2 -507.476} C_VEL
LIN {X 0,Y 608.472,Z 151.688,A -85,B 0,C 180,E1 -510.221,E2 -510.221} C_VEL
LIN {X 0,Y 608.469,Z 151.693,A -85,B 0,C 180,E1 -512.794,E2 -512.794} C_VEL
LIN {X 0,Y 608.438,Z 151.693,A -85,B 0,C 180,E1 -515.428,E2 -515.428} C_VEL
LIN {X 0,Y 608.436,Z 151.693,A -85,B 0,C 180,E1 -518.307,E2 -518.307} C_VEL
LIN {X 0,Y 608.452,Z 151.698,A -85,B 0,C 180,E1 -521.13,E2 -521.13} C_VEL
LIN {X 0,Y 608.454,Z 151.69,A -85,B 0,C 180,E1 -523.906,E2 -523.906} C_VEL
LIN {X 0,Y 608.453,Z 151.693,A -85,B 0,C 180,E1 -526.643,E2 -526.643} C_VEL
LIN {X 0,Y 608.465,Z 151.691,A -85,B 0,C 180,E1 -529.35,E2 -529.35} C_VEL
LIN {X 0,Y 608.408,Z 151.696,A -85,B 0,C 180,E1 -532.032,E2 -532.032} C_VEL
LIN {X 0,Y 608.459,Z 151.695,A -85,B 0,C 180,E1 -534.698,E2 -534.698} C_VEL
LIN {X 0,Y 608.469,Z 151.688,A -85,B 0,C 180,E1 -537.352,E2 -537.352} C_VEL
LIN {X 0,Y 608.477,Z 151.695,A -85,B 0,C 180,E1 -540,E2 -540} C_VEL
LIN {X 0,Y 608.468,Z 151.688,A -85,B 0,C 180,E1 -542.648,E2 -542.648} C_VEL
LIN {X 0,Y 608.455,Z 151.695,A -85,B 0,C 180,E1 -545.302,E2 -545.302} C_VEL
LIN {X 0,Y 608.409,Z 151.696,A -85,B 0,C 180,E1 -547.968,E2 -547.968} C_VEL
LIN {X 0,Y 608.431,Z 151.693,A -85,B 0,C 180,E1 -549.446,E2 -549.446} C_VEL
LIN {X 0,Y 607.759,Z 151.782,A -85,B 0,C 180,E1 -549.999,E2 -549.999} C_VEL
LIN {X 0,Y 604.918,Z 152.137,A -85,B 0,C 180,E1 -550.896,E2 -550.896} C_VEL
LIN {X 0,Y 602.522,Z 152.436,A -85,B 0,C 180,E1 -551.617,E2 -551.617} C_VEL
LIN {X 0,Y 601.494,Z 152.563,A -85,B 0,C 180,E1 -552.174,E2 -552.174} C_VEL
LIN {X 0,Y 601.41,Z 152.57,A -85,B 0,C 180,E1 -552.363,E2 -552.363} C_VEL
LIN {X 0,Y 601.432,Z 152.566,A -85,B 0,C 180,E1 -554.897,E2 -554.897} C_VEL
LIN {X 0,Y 601.43,Z 152.571,A -85,B 0,C 180,E1 -556.986,E2 -556.986} C_VEL
LIN {X 0,Y 601.389,Z 152.57,A -85,B 0,C 180,E1 -559.81,E2 -559.81} C_VEL
LIN {X 0,Y 601.412,Z 152.57,A -85,B 0,C 180,E1 -562.605,E2 -562.605} C_VEL
LIN {X 0,Y 601.387,Z 152.57,A -85,B 0,C 180,E1 -564.879,E2 -564.879} C_VEL
LIN {X 0,Y 601.412,Z 152.575,A -85,B 0,C 180,E1 -567.363,E2 -567.363} C_VEL
LIN {X 0,Y 601.428,Z 152.566,A -85,B 0,C 180,E1 -570.164,E2 -570.164} C_VEL
LIN {X 0,Y 601.42,Z 152.572,A -85,B 0,C 180,E1 -572.716,E2 -572.716} C_VEL
LIN {X 0,Y 601.372,Z 152.572,A -85,B 0,C 180,E1 -575.109,E2 -575.109} C_VEL
LIN {X 0,Y 601.394,Z 152.574,A -85,B 0,C 180,E1 -577.422,E2 -577.422} C_VEL
LIN {X 0,Y 601.4,Z 152.569,A -85,B 0,C 180,E1 -579.996,E2 -579.996} C_VEL
LIN {X 0,Y 601.407,Z 152.573,A -85,B 0,C 180,E1 -582.671,E2 -582.671} C_VEL
LIN {X 0,Y 601.426,Z 152.566,A -85,B 0,C 180,E1 -585.482,E2 -585.482} C_VEL
LIN {X 0,Y 601.413,Z 152.569,A -85,B 0,C 180,E1 -588.408,E2 -588.408} C_VEL
LIN {X 0,Y 601.385,Z 152.572,A -85,B 0,C 180,E1 -590.872,E2 -590.872} C_VEL
LIN {X 0,Y 601.387,Z 152.571,A -85,B 0,C 180,E1 -593.742,E2 -593.742} C_VEL
LIN {X 0,Y 601.378,Z 153.016,A -85,B 0,C 180,E1 -594.891,E2 -594.891} C_VEL
LIN {X 0,Y 601.411,Z 157.446,A -85,B 0,C 180,E1 -597.483,E2 -597.483} C_VEL
LIN {X 0,Y 601.402,Z 162.89,A -85,B 0,C 180,E1 -600.606,E2 -600.606} C_VEL
LIN {X 0,Y 601.386,Z 166.956,A -85,B 0,C 180,E1 -602.886,E2 -602.886} C_VEL
LIN {X 0,Y 601.384,Z 172.162,A -85,B 0,C 180,E1 -605.719,E2 -605.719} C_VEL
LIN {X 0,Y 601.354,Z 176.567,A -85,B 0,C 180,E1 -608.039,E2 -608.039} C_VEL
LIN {X 0,Y 601.351,Z 182.097,A -85,B 0,C 180,E1 -610.899,E2 -610.899} C_VEL
LIN {X 0,Y 601.338,Z 187.626,A -85,B 0,C 180,E1 -613.711,E2 -613.711} C_VEL
LIN {X 0,Y 601.323,Z 193.156,A -85,B 0,C 180,E1 -616.482,E2 -616.482} C_VEL
LIN {X 0,Y 601.34,Z 196.526,A -85,B 0,C 180,E1 -618.156,E2 -618.156} C_VEL
LIN {X 0,Y 601.599,Z 201.401,A -85,B 0,C 180,E1 -618.268,E2 -618.268} C_VEL
LIN {X 0,Y 601.558,Z 213.746,A -85,B 0,C 180,E1 -618.585,E2 -618.585} C_VEL
LIN {X 0,Y 601.5,Z 226.359,A -85,B 0,C 180,E1 -619.051,E2 -619.051} C_VEL
LIN {X 0,Y 601.447,Z 238.517,A -85,B 0,C 180,E1 -619.65,E2 -619.65} C_VEL
LIN {X 0,Y 601.461,Z 249.313,A -85,B 0,C 180,E1 -620.33,E2 -620.33} C_VEL
LIN {X 0,Y 601.435,Z 259.087,A -85,B 0,C 180,E1 -621.093,E2 -621.093} C_VEL
LIN {X 0,Y 601.407,Z 267.982,A -85,B 0,C 180,E1 -621.939,E2 -621.939} C_VEL
LIN {X 0,Y 601.406,Z 276.669,A -85,B 0,C 180,E1 -622.952,E2 -622.952} C_VEL
LIN {X 0,Y 601.361,Z 283.598,A -85,B 0,C 180,E1 -623.963,E2 -623.963} C_VEL
LIN {X 0,Y 601.344,Z 289.15,A -85,B 0,C 180,E1 -624.972,E2 -624.972} C_VEL
LIN {X 0,Y 601.347,Z 293.512,A -85,B 0,C 180,E1 -625.979,E2 -625.979} C_VEL
LIN {X 0,Y 601.344,Z 295.815,A -85,B 0,C 180,E1 -626.65,E2 -626.65} C_VEL
LIN {X 0,Y 601.324,Z 297.693,A -85,B 0,C 180,E1 -627.321,E2 -627.321} C_VEL
LIN {X 0,Y 601.343,Z 299.127,A -85,B 0,C 180,E1 -627.991,E2 -627.991} C_VEL
LIN {X 0,Y 601.339,Z 300.753,A -85,B 0,C 180,E1 -629.331,E2 -629.331} C_VEL
LIN {X 0,Y 601.336,Z 300.996,A -85,B 0,C 180,E1 -630,E2 -630} C_VEL
LIN {X 0,Y 601.339,Z 300.815,A -85,B 0,C 180,E1 -630.67,E2 -630.67} C_VEL
LIN {X 0,Y 601.343,Z 299.275,A -85,B 0,C 180,E1 -632.009,E2 -632.009} C_VEL
LIN {X 0,Y 601.326,Z 297.916,A -85,B 0,C 180,E1 -632.68,E2 -632.68} C_VEL
LIN {X 0,Y 601.368,Z 295.039,A -85,B 0,C 180,E1 -633.685,E2 -633.685} C_VEL
LIN {X 0,Y 601.337,Z 291.14,A -85,B 0,C 180,E1 -634.693,E2 -634.693} C_VEL
LIN {X 0,Y 601.373,Z 286.109,A -85,B 0,C 180,E1 -635.701,E2 -635.701} C_VEL
LIN {X 0,Y 601.382,Z 279.79,A -85,B 0,C 180,E1 -636.711,E2 -636.711} C_VEL
LIN {X 0,Y 601.396,Z 271.873,A -85,B 0,C 180,E1 -637.724,E2 -637.724} C_VEL
LIN {X 0,Y 601.437,Z 262.028,A -85,B 0,C 180,E1 -638.738,E2 -638.738} C_VEL
LIN {X 0,Y 601.445,Z 251.707,A -85,B 0,C 180,E1 -639.585,E2 -639.585} C_VEL
LIN {X 0,Y 601.441,Z 240.086,A -85,B 0,C 180,E1 -640.35,E2 -640.35} C_VEL
LIN {X 0,Y 601.483,Z 228.013,A -85,B 0,C 180,E1 -640.967,E2 -640.967} C_VEL
LIN {X 0,Y 601.549,Z 215.243,A -85,B 0,C 180,E1 -641.456,E2 -641.456} C_VEL
LIN {X 0,Y 601.602,Z 202.616,A -85,B 0,C 180,E1 -641.797,E2 -641.797} C_VEL
LIN {X 0,Y 601.329,Z 196.534,A -85,B 0,C 180,E1 -641.93,E2 -641.93} C_VEL
LIN {X 0,Y 601.306,Z 191.953,A -85,B 0,C 180,E1 -644.208,E2 -644.208} C_VEL
LIN {X 0,Y 601.336,Z 186.421,A -85,B 0,C 180,E1 -646.989,E2 -646.989} C_VEL
LIN {X 0,Y 601.331,Z 180.888,A -85,B 0,C 180,E1 -649.812,E2 -649.812} C_VEL
LIN {X 0,Y 601.368,Z 175.53,A -85,B 0,C 180,E1 -652.594,E2 -652.594} C_VEL
LIN {X 0,Y 601.347,Z 171.206,A -85,B 0,C 180,E1 -654.881,E2 -654.881} C_VEL
LIN {X 0,Y 601.395,Z 166.653,A -85,B 0,C 180,E1 -657.358,E2 -657.358} C_VEL
LIN {X 0,Y 601.381,Z 161.708,A -85,B 0,C 180,E1 -660.167,E2 -660.167} C_VEL
LIN {X 0,Y 601.39,Z 157.267,A -85,B 0,C 180,E1 -662.71,E2 -662.71} C_VEL
LIN {X 0,Y 601.394,Z 153.162,A -85,B 0,C 180,E1 -665.111,E2 -665.111} C_VEL
LIN {X 0,Y 601.38,Z 152.573,A -85,B 0,C 180,E1 -665.755,E2 -665.755} C_VEL
LIN {X 0,Y 601.38,Z 152.576,A -85,B 0,C 180,E1 -668.464,E2 -668.464} C_VEL
LIN {X 0,Y 601.395,Z 152.571,A -85,B 0,C 180,E1 -670.876,E2 -670.876} C_VEL
LIN {X 0,Y 601.43,Z 152.569,A -85,B 0,C 180,E1 -673.586,E2 -673.586} C_VEL
LIN {X 0,Y 601.431,Z 152.565,A -85,B 0,C 180,E1 -676.427,E2 -676.427} C_VEL
LIN {X 0,Y 601.415,Z 152.572,A -85,B 0,C 180,E1 -679.125,E2 -679.125} C_VEL
LIN {X 0,Y 601.397,Z 152.569,A -85,B 0,C 180,E1 -681.73,E2 -681.73} C_VEL
LIN {X 0,Y 601.38,Z 152.577,A -85,B 0,C 180,E1 -684.245,E2 -684.245} C_VEL
LIN {X 0,Y 601.412,Z 152.567,A -85,B 0,C 180,E1 -686.685,E2 -686.685} C_VEL
LIN {X 0,Y 601.414,Z 152.572,A -85,B 0,C 180,E1 -689.058,E2 -689.058} C_VEL
LIN {X 0,Y 601.427,Z 152.567,A -85,B 0,C 180,E1 -691.373,E2 -691.373} C_VEL
LIN {X 0,Y 601.416,Z 152.571,A -85,B 0,C 180,E1 -694.132,E2 -694.132} C_VEL
LIN {X 0,Y 601.379,Z 152.573,A -85,B 0,C 180,E1 -696.588,E2 -696.588} C_VEL
LIN {X 0,Y 601.426,Z 152.573,A -85,B 0,C 180,E1 -699.478,E2 -699.478} C_VEL
LIN {X 0,Y 601.386,Z 152.571,A -85,B 0,C 180,E1 -702.311,E2 -702.311} C_VEL
LIN {X 0,Y 601.412,Z 152.572,A -85,B 0,C 180,E1 -704.409,E2 -704.409} C_VEL
LIN {X 0,Y 601.419,Z 152.566,A -85,B 0,C 180,E1 -707.172,E2 -707.172} C_VEL
LIN {X 0,Y 601.421,Z 152.572,A -85,B 0,C 180,E1 -709.905,E2 -709.905} C_VEL
LIN {X 0,Y 601.371,Z 152.573,A -85,B 0,C 180,E1 -712.614,E2 -712.614} C_VEL
LIN {X 0,Y 601.409,Z 152.57,A -85,B 0,C 180,E1 -715.308,E2 -715.308} C_VEL
LIN {X 0,Y 601.414,Z 152.57,A -85,B 0,C 180,E1 -717.991,E2 -717.991} C_VEL
LIN {X 0,Y 601.449,Z 152.563,A -85,B 0,C 180,E1 -720.669,E2 -720.669} C_VEL
LIN {X 0,Y 601.431,Z 152.571,A -85,B 0,C 180,E1 -723.35,E2 -723.35} C_VEL
LIN {X 0,Y 601.374,Z 152.572,A -85,B 0,C 180,E1 -726.037,E2 -726.037} C_VEL
LIN {X 0,Y 601.408,Z 152.574,A -85,B 0,C 180,E1 -728.738,E2 -728.738} C_VEL
LIN {X 0,Y 601.407,Z 152.569,A -85,B 0,C 180,E1 -731.459,E2 -731.459} C_VEL
LIN {X 0,Y 601.422,Z 152.568,A -85,B 0,C 180,E1 -734.205,E2 -734.205} C_VEL
LIN {X 0,Y 601.433,Z 152.57,A -85,B 0,C 180,E1 -736.986,E2 -736.986} C_VEL
LIN {X 0,Y 601.392,Z 152.57,A -85,B 0,C 180,E1 -739.81,E2 -739.81} C_VEL
LIN {X 0,Y 601.415,Z 152.57,A -85,B 0,C 180,E1 -742.605,E2 -742.605} C_VEL
LIN {X 0,Y 601.385,Z 152.57,A -85,B 0,C 180,E1 -744.879,E2 -744.879} C_VEL
LIN {X 0,Y 601.411,Z 152.574,A -85,B 0,C 180,E1 -747.361,E2 -747.361} C_VEL
LIN {X 0,Y 601.43,Z 152.565,A -85,B 0,C 180,E1 -750.164,E2 -750.164} C_VEL
LIN {X 0,Y 601.42,Z 152.572,A -85,B 0,C 180,E1 -752.715,E2 -752.715} C_VEL
LIN {X 0,Y 601.375,Z 152.572,A -85,B 0,C 180,E1 -755.109,E2 -755.109} C_VEL
LIN {X 0,Y 601.395,Z 152.573,A -85,B 0,C 180,E1 -757.422,E2 -757.422} C_VEL
LIN {X 0,Y 601.382,Z 152.572,A -85,B 0,C 180,E1 -759.998,E2 -759.998} C_VEL
LIN {X 0,Y 601.408,Z 152.573,A -85,B 0,C 180,E1 -762.671,E2 -762.671} C_VEL
LIN {X 0,Y 601.4,Z 152.569,A -85,B 0,C 180,E1 -765.48,E2 -765.48} C_VEL
LIN {X 0,Y 601.415,Z 152.569,A -85,B 0,C 180,E1 -768.408,E2 -768.408} C_VEL
LIN {X 0,Y 601.387,Z 152.572,A -85,B 0,C 180,E1 -770.871,E2 -770.871} C_VEL
LIN {X 0,Y 601.388,Z 152.573,A -85,B 0,C 180,E1 -773.742,E2 -773.742} C_VEL
LIN {X 0,Y 601.428,Z 152.723,A -85,B 0,C 180,E1 -774.334,E2 -774.334} C_VEL
LIN {X 0,Y 601.525,Z 159.169,A -85,B 0,C 180,E1 -776.693,E2 -776.693} C_VEL
LIN {X 0,Y 601.467,Z 166.96,A -85,B 0,C 180,E1 -779.45,E2 -779.45} C_VEL
LIN {X 0,Y 601.445,Z 174.752,A -85,B 0,C 180,E1 -782.134,E2 -782.134} C_VEL
LIN {X 0,Y 601.428,Z 183.656,A -85,B 0,C 180,E1 -785.122,E2 -785.122} C_VEL
LIN {X 0,Y 601.42,Z 190.571,A -85,B 0,C 180,E1 -787.394,E2 -787.394} C_VEL
LIN {X 0,Y 601.403,Z 199.239,A -85,B 0,C 180,E1 -790.19,E2 -790.19} C_VEL
LIN {X 0,Y 601.377,Z 208.143,A -85,B 0,C 180,E1 -793.012,E2 -793.012} C_VEL
LIN {X 0,Y 601.368,Z 217.488,A -85,B 0,C 180,E1 -795.93,E2 -795.93} C_VEL
LIN {X 0,Y 601.364,Z 224.491,A -85,B 0,C 180,E1 -798.092,E2 -798.092} C_VEL
LIN {X 0,Y 601.601,Z 231.506,A -85,B 0,C 180,E1 -798.225,E2 -798.225} C_VEL
LIN {X 0,Y 601.555,Z 243.876,A -85,B 0,C 180,E1 -798.544,E2 -798.544} C_VEL
LIN {X 0,Y 601.493,Z 256.335,A -85,B 0,C 180,E1 -799.005,E2 -799.005} C_VEL
LIN {X 0,Y 601.458,Z 267.771,A -85,B 0,C 180,E1 -799.565,E2 -799.565} C_VEL
LIN {X 0,Y 601.468,Z 278.745,A -85,B 0,C 180,E1 -800.245,E2 -800.245} C_VEL
LIN {X 0,Y 601.435,Z 289.597,A -85,B 0,C 180,E1 -801.093,E2 -801.093} C_VEL
LIN {X 0,Y 601.407,Z 298.412,A -85,B 0,C 180,E1 -801.939,E2 -801.939} C_VEL
LIN {X 0,Y 601.388,Z 305.689,A -85,B 0,C 180,E1 -802.783,E2 -802.783} C_VEL
LIN {X 0,Y 601.375,Z 312.773,A -85,B 0,C 180,E1 -803.782,E2 -803.782} C_VEL
LIN {X 0,Y 601.373,Z 317.679,A -85,B 0,C 180,E1 -804.635,E2 -804.635} C_VEL
LIN {X 0,Y 601.354,Z 322.37,A -85,B 0,C 180,E1 -805.643,E2 -805.643} C_VEL
LIN {X 0,Y 601.344,Z 325.955,A -85,B 0,C 180,E1 -806.65,E2 -806.65} C_VEL
LIN {X 0,Y 601.325,Z 327.809,A -85,B 0,C 180,E1 -807.32,E2 -807.32} C_VEL
LIN {X 0,Y 601.343,Z 329.201,A -85,B 0,C 180,E1 -807.991,E2 -807.991} C_VEL
LIN {X 0,Y 601.339,Z 330.783,A -85,B 0,C 180,E1 -809.33,E2 -809.33} C_VEL
LIN {X 0,Y 601.335,Z 331,A -85,B 0,C 180,E1 -810,E2 -810} C_VEL
LIN {X 0,Y 601.347,Z 330.184,A -85,B 0,C 180,E1 -811.339,E2 -811.339} C_VEL
LIN {X 0,Y 601.343,Z 329.202,A -85,B 0,C 180,E1 -812.009,E2 -812.009} C_VEL
LIN {X 0,Y 601.325,Z 327.81,A -85,B 0,C 180,E1 -812.679,E2 -812.679} C_VEL
LIN {X 0,Y 601.368,Z 324.897,A -85,B 0,C 180,E1 -813.685,E2 -813.685} C_VEL
LIN {X 0,Y 601.336,Z 320.951,A -85,B 0,C 180,E1 -814.692,E2 -814.692} C_VEL
LIN {X 0,Y 601.372,Z 314.878,A -85,B 0,C 180,E1 -815.869,E2 -815.869} C_VEL
LIN {X 0,Y 601.381,Z 308.237,A -85,B 0,C 180,E1 -816.88,E2 -816.88} C_VEL
LIN {X 0,Y 601.4,Z 299.991,A -85,B 0,C 180,E1 -817.892,E2 -817.892} C_VEL
LIN {X 0,Y 601.436,Z 291.539,A -85,B 0,C 180,E1 -818.737,E2 -818.737} C_VEL
LIN {X 0,Y 601.446,Z 281.094,A -85,B 0,C 180,E1 -819.585,E2 -819.585} C_VEL
LIN {X 0,Y 601.442,Z 270.759,A -85,B 0,C 180,E1 -820.265,E2 -820.265} C_VEL
LIN {X 0,Y 601.479,Z 259.269,A -85,B 0,C 180,E1 -820.867,E2 -820.867} C_VEL
LIN {X 0,Y 601.526,Z 246.348,A -85,B 0,C 180,E1 -821.375,E2 -821.375} C_VEL
LIN {X 0,Y 601.605,Z 233.447,A -85,B 0,C 180,E1 -821.732,E2 -821.732} C_VEL
LIN {X 0,Y 601.494,Z 225.629,A -85,B 0,C 180,E1 -821.884,E2 -821.884} C_VEL
LIN {X 0,Y 601.335,Z 224.423,A -85,B 0,C 180,E1 -821.93,E2 -821.93} C_VEL
LIN {X 0,Y 601.343,Z 215.936,A -85,B 0,C 180,E1 -824.553,E2 -824.553} C_VEL
LIN {X 0,Y 601.393,Z 207.031,A -85,B 0,C 180,E1 -827.337,E2 -827.337} C_VEL
LIN {X 0,Y 601.387,Z 198.127,A -85,B 0,C 180,E1 -830.166,E2 -830.166} C_VEL
LIN {X 0,Y 601.428,Z 189.222,A -85,B 0,C 180,E1 -833.045,E2 -833.045} C_VEL
LIN {X 0,Y 601.431,Z 181.431,A -85,B 0,C 180,E1 -835.617,E2 -835.617} C_VEL
LIN {X 0,Y 601.441,Z 173.64,A -85,B 0,C 180,E1 -838.245,E2 -838.245} C_VEL
LIN {X 0,Y 601.47,Z 165.848,A -85,B 0,C 180,E1 -840.939,E2 -840.939} C_VEL
LIN {X 0,Y 601.525,Z 159.17,A -85,B 0,C 180,E1 -843.307,E2 -843.307} C_VEL
LIN {X 0,Y 601.417,Z 152.608,A -85,B 0,C 180,E1 -845.709,E2 -845.709} C_VEL
LIN {X 0,Y 601.395,Z 152.576,A -85,B 0,C 180,E1 -848.466,E2 -848.466} C_VEL
LIN {X 0,Y 601.401,Z 152.57,A -85,B 0,C 180,E1 -850.875,E2 -850.875} C_VEL
LIN {X 0,Y 601.428,Z 152.571,A -85,B 0,C 180,E1 -853.586,E2 -853.586} C_VEL
LIN {X 0,Y 601.429,Z 152.565,A -85,B 0,C 180,E1 -856.427,E2 -856.427} C_VEL
LIN {X 0,Y 601.41,Z 152.571,A -85,B 0,C 180,E1 -859.125,E2 -859.125} C_VEL
LIN {X 0,Y 601.393,Z 152.57,A -85,B 0,C 180,E1 -861.73,E2 -861.73} C_VEL
LIN {X 0,Y 601.381,Z 152.575,A -85,B 0,C 180,E1 -864.245,E2 -864.245} C_VEL
LIN {X 0,Y 601.412,Z 152.567,A -85,B 0,C 180,E1 -866.685,E2 -866.685} C_VEL
LIN {X 0,Y 601.416,Z 152.574,A -85,B 0,C 180,E1 -869.058,E2 -869.058} C_VEL
LIN {X 0,Y 601.423,Z 152.567,A -85,B 0,C 180,E1 -871.373,E2 -871.373} C_VEL
LIN {X 0,Y 601.415,Z 152.573,A -85,B 0,C 180,E1 -874.132,E2 -874.132} C_VEL
LIN {X 0,Y 601.375,Z 152.572,A -85,B 0,C 180,E1 -876.588,E2 -876.588} C_VEL
LIN {X 0,Y 601.428,Z 152.573,A -85,B 0,C 180,E1 -879.478,E2 -879.478} C_VEL
LIN {X 0,Y 601.39,Z 152.571,A -85,B 0,C 180,E1 -882.311,E2 -882.311} C_VEL
LIN {X 0,Y 601.411,Z 152.573,A -85,B 0,C 180,E1 -884.409,E2 -884.409} C_VEL
LIN {X 0,Y 601.419,Z 152.566,A -85,B 0,C 180,E1 -887.172,E2 -887.172} C_VEL
LIN {X 0,Y 601.415,Z 152.572,A -85,B 0,C 180,E1 -889.905,E2 -889.905} C_VEL
LIN {X 0,Y 601.372,Z 152.573,A -85,B 0,C 180,E1 -892.614,E2 -892.614} C_VEL
LIN {X 0,Y 601.412,Z 152.569,A -85,B 0,C 180,E1 -895.308,E2 -895.308} C_VEL
LIN {X 0,Y 601.42,Z 152.57,A -85,B 0,C 180,E1 -897.991,E2 -897.991} C_VEL
LIN {X 0,Y 601.447,Z 152.563,A -85,B 0,C 180,E1 -900.67,E2 -900.67} C_VEL
LIN {X 0,Y 601.431,Z 152.572,A -85,B 0,C 180,E1 -903.35,E2 -903.35} C_VEL
LIN {X 0,Y 601.371,Z 152.572,A -85,B 0,C 180,E1 -906.038,E2 -906.038} C_VEL
LIN {X 0,Y 601.409,Z 152.572,A -85,B 0,C 180,E1 -908.738,E2 -908.738} C_VEL
LIN {X 0,Y 601.408,Z 152.569,A -85,B 0,C 180,E1 -911.459,E2 -911.459} C_VEL
LIN {X 0,Y 601.41,Z 152.57,A -85,B 0,C 180,E1 -912.363,E2 -912.363} C_VEL
LIN {X 0,Y 600.744,Z 152.651,A -85,B 0,C 180,E1 -912.922,E2 -912.922} C_VEL
LIN {X 0,Y 597.896,Z 153.011,A -85,B 0,C 180,E1 -913.83,E2 -913.83} C_VEL
LIN {X 0,Y 595.487,Z 153.31,A -85,B 0,C 180,E1 -914.56,E2 -914.56} C_VEL
LIN {X 0,Y 594.448,Z 153.439,A -85,B 0,C 180,E1 -915.123,E2 -915.123} C_VEL
LIN {X 0,Y 594.361,Z 153.447,A -85,B 0,C 180,E1 -915.314,E2 -915.314} C_VEL
LIN {X 0,Y 594.386,Z 153.449,A -85,B 0,C 180,E1 -917.194,E2 -917.194} C_VEL
LIN {X 0,Y 594.364,Z 153.447,A -85,B 0,C 180,E1 -920.054,E2 -920.054} C_VEL
LIN {X 0,Y 594.347,Z 153.447,A -85,B 0,C 180,E1 -922.968,E2 -922.968} C_VEL
LIN {X 0,Y 594.361,Z 153.447,A -85,B 0,C 180,E1 -925.194,E2 -925.194} C_VEL
LIN {X 0,Y 594.385,Z 153.449,A -85,B 0,C 180,E1 -927.527,E2 -927.527} C_VEL
LIN {X 0,Y 594.385,Z 153.444,A -85,B 0,C 180,E1 -930.329,E2 -930.329} C_VEL
LIN {X 0,Y 594.375,Z 153.446,A -85,B 0,C 180,E1 -932.951,E2 -932.951} C_VEL
LIN {X 0,Y 594.321,Z 153.452,A -85,B 0,C 180,E1 -935.411,E2 -935.411} C_VEL
LIN {X 0,Y 594.359,Z 153.45,A -85,B 0,C 180,E1 -937.943,E2 -937.943} C_VEL
LIN {X 0,Y 594.372,Z 153.448,A -85,B 0,C 180,E1 -940.822,E2 -940.822} C_VEL
LIN {X 0,Y 594.365,Z 153.447,A -85,B 0,C 180,E1 -943.3,E2 -943.3} C_VEL
LIN {X 0,Y 594.368,Z 153.452,A -85,B 0,C 180,E1 -946.161,E2 -946.161} C_VEL
LIN {X 0,Y 594.371,Z 153.445,A -85,B 0,C 180,E1 -948.536,E2 -948.536} C_VEL
LIN {X 0,Y 594.359,Z 153.453,A -85,B 0,C 180,E1 -951.299,E2 -951.299} C_VEL
LIN {X 0,Y 594.341,Z 153.449,A -85,B 0,C 180,E1 -953.755,E2 -953.755} C_VEL
LIN {X 0,Y 594.306,Z 153.542,A -85,B 0,C 180,E1 -954.683,E2 -954.683} C_VEL
LIN {X 0,Y 594.339,Z 157.601,A -85,B 0,C 180,E1 -957.095,E2 -957.095} C_VEL
LIN {X 0,Y 594.313,Z 162.056,A -85,B 0,C 180,E1 -959.685,E2 -959.685} C_VEL
LIN {X 0,Y 594.334,Z 167.038,A -85,B 0,C 180,E1 -962.537,E2 -962.537} C_VEL
LIN {X 0,Y 594.296,Z 171.07,A -85,B 0,C 180,E1 -964.804,E2 -964.804} C_VEL
LIN {X 0,Y 594.274,Z 176.568,A -85,B 0,C 180,E1 -967.763,E2 -967.763} C_VEL
LIN {X 0,Y 594.244,Z 180.715,A -85,B 0,C 180,E1 -969.942,E2 -969.942} C_VEL
LIN {X 0,Y 594.235,Z 184.863,A -85,B 0,C 180,E1 -972.092,E2 -972.092} C_VEL
LIN {X 0,Y 594.254,Z 190.392,A -85,B 0,C 180,E1 -974.919,E2 -974.919} C_VEL
LIN {X 0,Y 594.262,Z 196.527,A -85,B 0,C 180,E1 -978.013,E2 -978.013} C_VEL
LIN {X 0,Y 594.655,Z 201.428,A -85,B 0,C 180,E1 -978.129,E2 -978.129} C_VEL
LIN {X 0,Y 594.595,Z 213.839,A -85,B 0,C 180,E1 -978.452,E2 -978.452} C_VEL
LIN {X 0,Y 594.526,Z 226.374,A -85,B 0,C 180,E1 -978.921,E2 -978.921} C_VEL
LIN {X 0,Y 594.463,Z 238.53,A -85,B 0,C 180,E1 -979.527,E2 -979.527} C_VEL
LIN {X 0,Y 594.44,Z 249.318,A -85,B 0,C 180,E1 -980.215,E2 -980.215} C_VEL
LIN {X 0,Y 594.404,Z 259.094,A -85,B 0,C 180,E1 -980.987,E2 -980.987} C_VEL
LIN {X 0,Y 594.366,Z 267.987,A -85,B 0,C 180,E1 -981.843,E2 -981.843} C_VEL
LIN {X 0,Y 594.345,Z 276.673,A -85,B 0,C 180,E1 -982.868,E2 -982.868} C_VEL
LIN {X 0,Y 594.29,Z 283.601,A -85,B 0,C 180,E1 -983.89,E2 -983.89} C_VEL
LIN {X 0,Y 594.253,Z 289.152,A -85,B 0,C 180,E1 -984.911,E2 -984.911} C_VEL
LIN {X 0,Y 594.263,Z 293.514,A -85,B 0,C 180,E1 -985.931,E2 -985.931} C_VEL
LIN {X 0,Y 594.267,Z 295.817,A -85,B 0,C 180,E1 -986.61,E2 -986.61} C_VEL
LIN {X 0,Y 594.225,Z 297.695,A -85,B 0,C 180,E1 -987.289,E2 -987.289} C_VEL
LIN {X 0,Y 594.242,Z 299.127,A -85,B 0,C 180,E1 -987.967,E2 -987.967} C_VEL
LIN {X 0,Y 594.24,Z 300.753,A -85,B 0,C 180,E1 -989.323,E2 -989.323} C_VEL
LIN {X 0,Y 594.236,Z 300.996,A -85,B 0,C 180,E1 -990,E2 -990} C_VEL
LIN {X 0,Y 594.239,Z 300.815,A -85,B 0,C 180,E1 -990.678,E2 -990.678} C_VEL
LIN {X 0,Y 594.242,Z 299.275,A -85,B 0,C 180,E1 -992.033,E2 -992.033} C_VEL
LIN {X 0,Y 594.226,Z 297.914,A -85,B 0,C 180,E1 -992.712,E2 -992.712} C_VEL
LIN {X 0,Y 594.289,Z 295.037,A -85,B 0,C 180,E1 -993.729,E2 -993.729} C_VEL
LIN {X 0,Y 594.241,Z 291.138,A -85,B 0,C 180,E1 -994.749,E2 -994.749} C_VEL
LIN {X 0,Y 594.3,Z 286.106,A -85,B 0,C 180,E1 -995.769,E2 -995.769} C_VEL
LIN {X 0,Y 594.316,Z 279.786,A -85,B 0,C 180,E1 -996.791,E2 -996.791} C_VEL
LIN {X 0,Y 594.346,Z 271.868,A -85,B 0,C 180,E1 -997.816,E2 -997.816} C_VEL
LIN {X 0,Y 594.381,Z 262.022,A -85,B 0,C 180,E1 -998.842,E2 -998.842} C_VEL
LIN {X 0,Y 594.428,Z 251.701,A -85,B 0,C 180,E1 -999.7,E2 -999.7} C_VEL
LIN {X 0,Y 594.457,Z 240.075,A -85,B 0,C 180,E1 -1000.473,E2 -1000.473} C_VEL
LIN {X 0,Y 594.502,Z 228.961,A -85,B 0,C 180,E1 -1001.055,E2 -1001.055} C_VEL
LIN {X 0,Y 594.587,Z 216.554,A -85,B 0,C 180,E1 -1001.548,E2 -1001.548} C_VEL
LIN {X 0,Y 594.661,Z 203.507,A -85,B 0,C 180,E1 -1001.915,E2 -1001.915} C_VEL
LIN {X 0,Y 594.478,Z 198.171,A -85,B 0,C 180,E1 -1002.027,E2 -1002.027} C_VEL
LIN {X 0,Y 594.24,Z 196.533,A -85,B 0,C 180,E1 -1002.075,E2 -1002.075} C_VEL
LIN {X 0,Y 594.241,Z 190.569,A -85,B 0,C 180,E1 -1005.081,E2 -1005.081} C_VEL
LIN {X 0,Y 594.242,Z 186.42,A -85,B 0,C 180,E1 -1007.198,E2 -1007.198} C_VEL
LIN {X 0,Y 594.264,Z 182.27,A -85,B 0,C 180,E1 -1009.338,E2 -1009.338} C_VEL
LIN {X 0,Y 594.284,Z 178.121,A -85,B 0,C 180,E1 -1011.507,E2 -1011.507} C_VEL
LIN {X 0,Y 594.281,Z 173.971,A -85,B 0,C 180,E1 -1013.709,E2 -1013.709} C_VEL
LIN {X 0,Y 594.316,Z 169.769,A -85,B 0,C 180,E1 -1016.008,E2 -1016.008} C_VEL
LIN {X 0,Y 594.313,Z 165.86,A -85,B 0,C 180,E1 -1018.23,E2 -1018.23} C_VEL
LIN {X 0,Y 594.304,Z 161.788,A -85,B 0,C 180,E1 -1020.564,E2 -1020.564} C_VEL
LIN {X 0,Y 594.34,Z 157.672,A -85,B 0,C 180,E1 -1022.953,E2 -1022.953} C_VEL
LIN {X 0,Y 594.313,Z 153.532,A -85,B 0,C 180,E1 -1025.412,E2 -1025.412} C_VEL
LIN {X 0,Y 594.354,Z 153.447,A -85,B 0,C 180,E1 -1027.604,E2 -1027.604} C_VEL
LIN {X 0,Y 594.357,Z 153.452,A -85,B 0,C 180,E1 -1030.568,E2 -1030.568} C_VEL
LIN {X 0,Y 594.367,Z 153.446,A -85,B 0,C 180,E1 -1033.3,E2 -1033.3} C_VEL
LIN {X 0,Y 594.362,Z 153.446,A -85,B 0,C 180,E1 -1036.161,E2 -1036.161} C_VEL
LIN {X 0,Y 594.382,Z 153.445,A -85,B 0,C 180,E1 -1038.536,E2 -1038.536} C_VEL
LIN {X 0,Y 594.364,Z 153.446,A -85,B 0,C 180,E1 -1041.298,E2 -1041.298} C_VEL
LIN {X 0,Y 594.342,Z 153.451,A -85,B 0,C 180,E1 -1043.755,E2 -1043.755} C_VEL
LIN {X 0,Y 594.362,Z 153.448,A -85,B 0,C 180,E1 -1046.237,E2 -1046.237} C_VEL
LIN {X 0,Y 594.37,Z 153.445,A -85,B 0,C 180,E1 -1048.65,E2 -1048.65} C_VEL
LIN {X 0,Y 594.383,Z 153.45,A -85,B 0,C 180,E1 -1051.042,E2 -1051.042} C_VEL
LIN {X 0,Y 594.389,Z 153.444,A -85,B 0,C 180,E1 -1053.977,E2 -1053.977} C_VEL
LIN {X 0,Y 594.37,Z 153.449,A -85,B 0,C 180,E1 -1056.295,E2 -1056.295} C_VEL
LIN {X 0,Y 594.399,Z 153.444,A -85,B 0,C 180,E1 -1059.224,E2 -1059.224} C_VEL
LIN {X 0,Y 594.341,Z 153.448,A -85,B 0,C 180,E1 -1062.095,E2 -1062.095} C_VEL
LIN {X 0,Y 594.365,Z 153.447,A -85,B 0,C 180,E1 -1064.219,E2 -1064.219} C_VEL
LIN {X 0,Y 594.379,Z 153.451,A -85,B 0,C 180,E1 -1066.321,E2 -1066.321} C_VEL
LIN {X 0,Y 594.377,Z 153.444,A -85,B 0,C 180,E1 -1069.095,E2 -1069.095} C_VEL
LIN {X 0,Y 594.348,Z 153.45,A -85,B 0,C 180,E1 -1071.842,E2 -1071.842} C_VEL
LIN {X 0,Y 594.373,Z 153.447,A -85,B 0,C 180,E1 -1074.572,E2 -1074.572} C_VEL
LIN {X 0,Y 594.401,Z 153.441,A -85,B 0,C 180,E1 -1077.289,E2 -1077.289} C_VEL
LIN {X 0,Y 594.415,Z 153.446,A -85,B 0,C 180,E1 -1080,E2 -1080} C_VEL
LIN {X 0,Y 594.404,Z 153.44,A -85,B 0,C 180,E1 -1082.711,E2 -1082.711} C_VEL
LIN {X 0,Y 594.384,Z 153.447,A -85,B 0,C 180,E1 -1085.428,E2 -1085.428} C_VEL
LIN {X 0,Y 594.345,Z 153.449,A -85,B 0,C 180,E1 -1088.158,E2 -1088.158} C_VEL
LIN {X 0,Y 594.39,Z 153.442,A -85,B 0,C 180,E1 -1091.074,E2 -1091.074} C_VEL
LIN {X 0,Y 594.378,Z 153.45,A -85,B 0,C 180,E1 -1093.679,E2 -1093.679} C_VEL
LIN {X 0,Y 594.397,Z 153.443,A -85,B 0,C 180,E1 -1096.72,E2 -1096.72} C_VEL
LIN {X 0,Y 594.361,Z 153.448,A -85,B 0,C 180,E1 -1099.335,E2 -1099.335} C_VEL
LIN {X 0,Y 594.349,Z 153.447,A -85,B 0,C 180,E1 -1101.504,E2 -1101.504} C_VEL
LIN {X 0,Y 594.39,Z 153.444,A -85,B 0,C 180,E1 -1104.446,E2 -1104.446} C_VEL
LIN {X 0,Y 594.376,Z 153.451,A -85,B 0,C 180,E1 -1107.461,E2 -1107.461} C_VEL
LIN {X 0,Y 594.388,Z 153.444,A -85,B 0,C 180,E1 -1110.328,E2 -1110.328} C_VEL
LIN {X 0,Y 594.377,Z 153.446,A -85,B 0,C 180,E1 -1112.95,E2 -1112.95} C_VEL
LIN {X 0,Y 594.324,Z 153.451,A -85,B 0,C 180,E1 -1115.411,E2 -1115.411} C_VEL
LIN {X 0,Y 594.346,Z 153.452,A -85,B 0,C 180,E1 -1117.944,E2 -1117.944} C_VEL
LIN {X 0,Y 594.373,Z 153.447,A -85,B 0,C 180,E1 -1120.821,E2 -1120.821} C_VEL
LIN {X 0,Y 594.367,Z 153.447,A -85,B 0,C 180,E1 -1123.3,E2 -1123.3} C_VEL
LIN {X 0,Y 594.362,Z 153.452,A -85,B 0,C 180,E1 -1126.161,E2 -1126.161} C_VEL
LIN {X 0,Y 594.372,Z 153.446,A -85,B 0,C 180,E1 -1128.535,E2 -1128.535} C_VEL
LIN {X 0,Y 594.361,Z 153.452,A -85,B 0,C 180,E1 -1131.299,E2 -1131.299} C_VEL
LIN {X 0,Y 594.367,Z 153.604,A -85,B 0,C 180,E1 -1134.175,E2 -1134.175} C_VEL
LIN {X 0,Y 594.498,Z 158.075,A -85,B 0,C 180,E1 -1135.845,E2 -1135.845} C_VEL
LIN {X 0,Y 594.48,Z 164.966,A -85,B 0,C 180,E1 -1138.342,E2 -1138.342} C_VEL
LIN {X 0,Y 594.454,Z 172.597,A -85,B 0,C 180,E1 -1141.03,E2 -1141.03} C_VEL
LIN {X 0,Y 594.399,Z 179.204,A -85,B 0,C 180,E1 -1143.301,E2 -1143.301} C_VEL
LIN {X 0,Y 594.415,Z 187.01,A -85,B 0,C 180,E1 -1145.931,E2 -1145.931} C_VEL
LIN {X 0,Y 594.37,Z 194.787,A -85,B 0,C 180,E1 -1148.497,E2 -1148.497} C_VEL
LIN {X 0,Y 594.322,Z 203.691,A -85,B 0,C 180,E1 -1151.38,E2 -1151.38} C_VEL
LIN {X 0,Y 594.295,Z 212.596,A -85,B 0,C 180,E1 -1154.217,E2 -1154.217} C_VEL
LIN {X 0,Y 594.264,Z 221.5,A -85,B 0,C 180,E1 -1157.015,E2 -1157.015} C_VEL
LIN {X 0,Y 594.273,Z 224.491,A -85,B 0,C 180,E1 -1157.947,E2 -1157.947} C_VEL
LIN {X 0,Y 594.663,Z 229.223,A -85,B 0,C 180,E1 -1158.042,E2 -1158.042} C_VEL
LIN {X 0,Y 594.622,Z 242.491,A -85,B 0,C 180,E1 -1158.365,E2 -1158.365} C_VEL
LIN {X 0,Y 594.53,Z 254.664,A -85,B 0,C 180,E1 -1158.802,E2 -1158.802} C_VEL
LIN {X 0,Y 594.469,Z 266.205,A -85,B 0,C 180,E1 -1159.355,E2 -1159.355} C_VEL
LIN {X 0,Y 594.452,Z 277.473,A -85,B 0,C 180,E1 -1160.043,E2 -1160.043} C_VEL
LIN {X 0,Y 594.406,Z 287.645,A -85,B 0,C 180,E1 -1160.815,E2 -1160.815} C_VEL
LIN {X 0,Y 594.372,Z 296.786,A -85,B 0,C 180,E1 -1161.671,E2 -1161.671} C_VEL
LIN {X 0,Y 594.316,Z 305.69,A -85,B 0,C 180,E1 -1162.697,E2 -1162.697} C_VEL
LIN {X 0,Y 594.281,Z 312.169,A -85,B 0,C 180,E1 -1163.615,E2 -1163.615} C_VEL
LIN {X 0,Y 594.289,Z 317.679,A -85,B 0,C 180,E1 -1164.571,E2 -1164.571} C_VEL
LIN {X 0,Y 594.27,Z 322.37,A -85,B 0,C 180,E1 -1165.591,E2 -1165.591} C_VEL
LIN {X 0,Y 594.267,Z 325.955,A -85,B 0,C 180,E1 -1166.61,E2 -1166.61} C_VEL
LIN {X 0,Y 594.226,Z 327.809,A -85,B 0,C 180,E1 -1167.288,E2 -1167.288} C_VEL
LIN {X 0,Y 594.242,Z 329.201,A -85,B 0,C 180,E1 -1167.967,E2 -1167.967} C_VEL
LIN {X 0,Y 594.239,Z 330.784,A -85,B 0,C 180,E1 -1169.322,E2 -1169.322} C_VEL
LIN {X 0,Y 594.236,Z 331,A -85,B 0,C 180,E1 -1170,E2 -1170} C_VEL
LIN {X 0,Y 594.247,Z 330.184,A -85,B 0,C 180,E1 -1171.355,E2 -1171.355} C_VEL
LIN {X 0,Y 594.242,Z 329.202,A -85,B 0,C 180,E1 -1172.033,E2 -1172.033} C_VEL
LIN {X 0,Y 594.225,Z 327.81,A -85,B 0,C 180,E1 -1172.711,E2 -1172.711} C_VEL
LIN {X 0,Y 594.289,Z 324.897,A -85,B 0,C 180,E1 -1173.729,E2 -1173.729} C_VEL
LIN {X 0,Y 594.241,Z 320.951,A -85,B 0,C 180,E1 -1174.749,E2 -1174.749} C_VEL
LIN {X 0,Y 594.305,Z 314.878,A -85,B 0,C 180,E1 -1175.939,E2 -1175.939} C_VEL
LIN {X 0,Y 594.308,Z 308.237,A -85,B 0,C 180,E1 -1176.962,E2 -1176.962} C_VEL
LIN {X 0,Y 594.359,Z 299.991,A -85,B 0,C 180,E1 -1177.986,E2 -1177.986} C_VEL
LIN {X 0,Y 594.382,Z 291.539,A -85,B 0,C 180,E1 -1178.842,E2 -1178.842} C_VEL
LIN {X 0,Y 594.431,Z 281.095,A -85,B 0,C 180,E1 -1179.699,E2 -1179.699} C_VEL
LIN {X 0,Y 594.445,Z 270.76,A -85,B 0,C 180,E1 -1180.387,E2 -1180.387} C_VEL
LIN {X 0,Y 594.498,Z 258.787,A -85,B 0,C 180,E1 -1181.018,E2 -1181.018} C_VEL
LIN {X 0,Y 594.559,Z 246.503,A -85,B 0,C 180,E1 -1181.505,E2 -1181.505} C_VEL
LIN {X 0,Y 594.674,Z 233.447,A -85,B 0,C 180,E1 -1181.871,E2 -1181.871} C_VEL
LIN {X 0,Y 594.412,Z 225.629,A -85,B 0,C 180,E1 -1182.028,E2 -1182.028} C_VEL
LIN {X 0,Y 594.277,Z 224.423,A -85,B 0,C 180,E1 -1182.074,E2 -1182.074} C_VEL
LIN {X 0,Y 594.292,Z 215.936,A -85,B 0,C 180,E1 -1184.729,E2 -1184.729} C_VEL
LIN {X 0,Y 594.321,Z 207.031,A -85,B 0,C 180,E1 -1187.55,E2 -1187.55} C_VEL
LIN {X 0,Y 594.358,Z 198.127,A -85,B 0,C 180,E1 -1190.415,E2 -1190.415} C_VEL
LIN {X 0,Y 594.371,Z 189.222,A -85,B 0,C 180,E1 -1193.335,E2 -1193.335} C_VEL
LIN {X 0,Y 594.402,Z 181.187,A -85,B 0,C 180,E1 -1196.025,E2 -1196.025} C_VEL
LIN {X 0,Y 594.433,Z 173.675,A -85,B 0,C 180,E1 -1198.596,E2 -1198.596} C_VEL
LIN {X 0,Y 594.465,Z 165.848,A -85,B 0,C 180,E1 -1201.344,E2 -1201.344} C_VEL
LIN {X 0,Y 594.496,Z 159.17,A -85,B 0,C 180,E1 -1203.753,E2 -1203.753} C_VEL
LIN {X 0,Y 594.545,Z 154.718,A -85,B 0,C 180,E1 -1205.395,E2 -1205.395} C_VEL
LIN {X 0,Y 594.355,Z 153.452,A -85,B 0,C 180,E1 -1205.93,E2 -1205.93} C_VEL
LIN {X 0,Y 594.359,Z 153.451,A -85,B 0,C 180,E1 -1208.807,E2 -1208.807} C_VEL
LIN {X 0,Y 594.38,Z 153.449,A -85,B 0,C 180,E1 -1211.848,E2 -1211.848} C_VEL
LIN {X 0,Y 594.355,Z 153.447,A -85,B 0,C 180,E1 -1214.808,E2 -1214.808} C_VEL
LIN {X 0,Y 594.363,Z 153.447,A -85,B 0,C 180,E1 -1217.624,E2 -1217.624} C_VEL
LIN {X 0,Y 594.365,Z 153.449,A -85,B 0,C 180,E1 -1220.319,E2 -1220.319} C_VEL
LIN {X 0,Y 594.327,Z 153.45,A -85,B 0,C 180,E1 -1222.909,E2 -1222.909} C_VEL
LIN {X 0,Y 594.374,Z 153.45,A -85,B 0,C 180,E1 -1225.862,E2 -1225.862} C_VEL
LIN {X 0,Y 594.37,Z 153.446,A -85,B 0,C 180,E1 -1228.65,E2 -1228.65} C_VEL
LIN {X 0,Y 594.38,Z 153.448,A -85,B 0,C 180,E1 -1231.042,E2 -1231.042} C_VEL
LIN {X 0,Y 594.387,Z 153.446,A -85,B 0,C 180,E1 -1233.976,E2 -1233.976} C_VEL
LIN {X 0,Y 594.367,Z 153.448,A -85,B 0,C 180,E1 -1236.295,E2 -1236.295} C_VEL
LIN {X 0,Y 594.401,Z 153.445,A -85,B 0,C 180,E1 -1239.224,E2 -1239.224} C_VEL
LIN {X 0,Y 594.349,Z 153.447,A -85,B 0,C 180,E1 -1242.095,E2 -1242.095} C_VEL
LIN {X 0,Y 594.364,Z 153.448,A -85,B 0,C 180,E1 -1244.219,E2 -1244.219} C_VEL
LIN {X 0,Y 594.377,Z 153.451,A -85,B 0,C 180,E1 -1246.321,E2 -1246.321} C_VEL
LIN {X 0,Y 594.375,Z 153.445,A -85,B 0,C 180,E1 -1249.095,E2 -1249.095} C_VEL
LIN {X 0,Y 594.345,Z 153.449,A -85,B 0,C 180,E1 -1251.842,E2 -1251.842} C_VEL
LIN {X 0,Y 594.38,Z 153.447,A -85,B 0,C 180,E1 -1254.572,E2 -1254.572} C_VEL
LIN {X 0,Y 594.402,Z 153.441,A -85,B 0,C 180,E1 -1257.289,E2 -1257.289} C_VEL
LIN {X 0,Y 594.414,Z 153.447,A -85,B 0,C 180,E1 -1260,E2 -1260} C_VEL
LIN {X 0,Y 594.402,Z 153.441,A -85,B 0,C 180,E1 -1262.711,E2 -1262.711} C_VEL
LIN {X 0,Y 594.377,Z 153.447,A -85,B 0,C 180,E1 -1265.428,E2 -1265.428} C_VEL
LIN {X 0,Y 594.346,Z 153.45,A -85,B 0,C 180,E1 -1268.158,E2 -1268.158} C_VEL
LIN {X 0,Y 594.389,Z 153.442,A -85,B 0,C 180,E1 -1271.075,E2 -1271.075} C_VEL
LIN {X 0,Y 594.378,Z 153.451,A -85,B 0,C 180,E1 -1273.679,E2 -1273.679} C_VEL
LIN {X 0,Y 594.361,Z 153.447,A -85,B 0,C 180,E1 -1275.314,E2 -1275.314} C_VEL
LIN {X 0,Y 593.684,Z 153.533,A -85,B 0,C 180,E1 -1275.88,E2 -1275.88} C_VEL
LIN {X 0,Y 590.816,Z 153.891,A -85,B 0,C 180,E1 -1276.798,E2 -1276.798} C_VEL
LIN {X 0,Y 588.405,Z 154.19,A -85,B 0,C 180,E1 -1277.537,E2 -1277.537} C_VEL
LIN {X 0,Y 587.383,Z 154.316,A -85,B 0,C 180,E1 -1278.107,E2 -1278.107} C_VEL
LIN {X 0,Y 587.306,Z 154.326,A -85,B 0,C 180,E1 -1278.3,E2 -1278.3} C_VEL
LIN {X 0,Y 587.329,Z 154.323,A -85,B 0,C 180,E1 -1281.038,E2 -1281.038} C_VEL
LIN {X 0,Y 587.324,Z 154.329,A -85,B 0,C 180,E1 -1284.007,E2 -1284.007} C_VEL
LIN {X 0,Y 587.338,Z 154.321,A -85,B 0,C 180,E1 -1286.279,E2 -1286.279} C_VEL
LIN {X 0,Y 587.348,Z 154.327,A -85,B 0,C 180,E1 -1289.134,E2 -1289.134} C_VEL
LIN {X 0,Y 587.345,Z 154.32,A -85,B 0,C 180,E1 -1291.836,E2 -1291.836} C_VEL
LIN {X 0,Y 587.338,Z 154.327,A -85,B 0,C 180,E1 -1294.347,E2 -1294.347} C_VEL
LIN {X 0,Y 587.313,Z 154.331,A -85,B 0,C 180,E1 -1297.61,E2 -1297.61} C_VEL
LIN {X 0,Y 587.307,Z 154.324,A -85,B 0,C 180,E1 -1300.255,E2 -1300.255} C_VEL
LIN {X 0,Y 587.314,Z 154.327,A -85,B 0,C 180,E1 -1303.119,E2 -1303.119} C_VEL
LIN {X 0,Y 587.323,Z 154.327,A -85,B 0,C 180,E1 -1306.05,E2 -1306.05} C_VEL
LIN {X 0,Y 587.33,Z 154.322,A -85,B 0,C 180,E1 -1308.926,E2 -1308.926} C_VEL
LIN {X 0,Y 587.306,Z 154.331,A -85,B 0,C 180,E1 -1311.519,E2 -1311.519} C_VEL
LIN {X 0,Y 587.27,Z 154.33,A -85,B 0,C 180,E1 -1314.099,E2 -1314.099} C_VEL
LIN {X 0,Y 587.256,Z 154.334,A -85,B 0,C 180,E1 -1314.468,E2 -1314.468} C_VEL
LIN {X 0,Y 587.267,Z 156.231,A -85,B 0,C 180,E1 -1315.774,E2 -1315.774} C_VEL
LIN {X 0,Y 587.298,Z 160.354,A -85,B 0,C 180,E1 -1318.229,E2 -1318.229} C_VEL
LIN {X 0,Y 587.279,Z 164.869,A -85,B 0,C 180,E1 -1320.88,E2 -1320.88} C_VEL
LIN {X 0,Y 587.253,Z 169.834,A -85,B 0,C 180,E1 -1323.718,E2 -1323.718} C_VEL
LIN {X 0,Y 587.216,Z 173.854,A -85,B 0,C 180,E1 -1325.989,E2 -1325.989} C_VEL
LIN {X 0,Y 587.189,Z 177.952,A -85,B 0,C 180,E1 -1328.221,E2 -1328.221} C_VEL
LIN {X 0,Y 587.202,Z 183.481,A -85,B 0,C 180,E1 -1331.147,E2 -1331.147} C_VEL
LIN {X 0,Y 587.159,Z 189.011,A -85,B 0,C 180,E1 -1334.02,E2 -1334.02} C_VEL
LIN {X 0,Y 587.166,Z 193.158,A -85,B 0,C 180,E1 -1336.15,E2 -1336.15} C_VEL
LIN {X 0,Y 587.147,Z 196.528,A -85,B 0,C 180,E1 -1337.865,E2 -1337.865} C_VEL
LIN {X 0,Y 587.734,Z 201.456,A -85,B 0,C 180,E1 -1337.987,E2 -1337.987} C_VEL
LIN {X 0,Y 587.647,Z 213.954,A -85,B 0,C 180,E1 -1338.317,E2 -1338.317} C_VEL
LIN {X 0,Y 587.559,Z 226.717,A -85,B 0,C 180,E1 -1338.803,E2 -1338.803} C_VEL
LIN {X 0,Y 587.482,Z 238.542,A -85,B 0,C 180,E1 -1339.401,E2 -1339.401} C_VEL
LIN {X 0,Y 587.431,Z 249.324,A -85,B 0,C 180,E1 -1340.097,E2 -1340.097} C_VEL
LIN {X 0,Y 587.357,Z 259.099,A -85,B 0,C 180,E1 -1340.878,E2 -1340.878} C_VEL
LIN {X 0,Y 587.302,Z 267.993,A -85,B 0,C 180,E1 -1341.744,E2 -1341.744} C_VEL
LIN {X 0,Y 587.274,Z 276.677,A -85,B 0,C 180,E1 -1342.782,E2 -1342.782} C_VEL
LIN {X 0,Y 587.214,Z 283.605,A -85,B 0,C 180,E1 -1343.817,E2 -1343.817} C_VEL
LIN {X 0,Y 587.167,Z 289.155,A -85,B 0,C 180,E1 -1344.85,E2 -1344.85} C_VEL
LIN {X 0,Y 587.182,Z 293.516,A -85,B 0,C 180,E1 -1345.882,E2 -1345.882} C_VEL
LIN {X 0,Y 587.194,Z 295.82,A -85,B 0,C 180,E1 -1346.569,E2 -1346.569} C_VEL
LIN {X 0,Y 587.131,Z 297.697,A -85,B 0,C 180,E1 -1347.256,E2 -1347.256} C_VEL
LIN {X 0,Y 587.141,Z 299.127,A -85,B 0,C 180,E1 -1347.942,E2 -1347.942} C_VEL
LIN {X 0,Y 587.14,Z 300.754,A -85,B 0,C 180,E1 -1349.314,E2 -1349.314} C_VEL
LIN {X 0,Y 587.137,Z 300.996,A -85,B 0,C 180,E1 -1350,E2 -1350} C_VEL
LIN {X 0,Y 587.14,Z 300.815,A -85,B 0,C 180,E1 -1350.686,E2 -1350.686} C_VEL
LIN {X 0,Y 587.141,Z 299.273,A -85,B 0,C 180,E1 -1352.058,E2 -1352.058} C_VEL
LIN {X 0,Y 587.133,Z 297.912,A -85,B 0,C 180,E1 -1352.745,E2 -1352.745} C_VEL
LIN {X 0,Y 587.213,Z 295.035,A -85,B 0,C 180,E1 -1353.774,E2 -1353.774} C_VEL
LIN {X 0,Y 587.147,Z 291.135,A -85,B 0,C 180,E1 -1354.806,E2 -1354.806} C_VEL
LIN {X 0,Y 587.23,Z 286.104,A -85,B 0,C 180,E1 -1355.839,E2 -1355.839} C_VEL
LIN {X 0,Y 587.23,Z 279.783,A -85,B 0,C 180,E1 -1356.874,E2 -1356.874} C_VEL
LIN {X 0,Y 587.288,Z 271.864,A -85,B 0,C 180,E1 -1357.91,E2 -1357.91} C_VEL
LIN {X 0,Y 587.343,Z 262.016,A -85,B 0,C 180,E1 -1358.949,E2 -1358.949} C_VEL
LIN {X 0,Y 587.41,Z 251.695,A -85,B 0,C 180,E1 -1359.817,E2 -1359.817} C_VEL
LIN {X 0,Y 587.445,Z 241.487,A -85,B 0,C 180,E1 -1360.512,E2 -1360.512} C_VEL
LIN {X 0,Y 587.526,Z 229.796,A -85,B 0,C 180,E1 -1361.147,E2 -1361.147} C_VEL
LIN {X 0,Y 587.623,Z 217.784,A -85,B 0,C 180,E1 -1361.644,E2 -1361.644} C_VEL
LIN {X 0,Y 587.699,Z 204.399,A -85,B 0,C 180,E1 -1362.036,E2 -1362.036} C_VEL
LIN {X 0,Y 587.515,Z 198.854,A -85,B 0,C 180,E1 -1362.158,E2 -1362.158} C_VEL
LIN {X 0,Y 587.143,Z 196.532,A -85,B 0,C 180,E1 -1362.223,E2 -1362.223} C_VEL
LIN {X 0,Y 587.145,Z 191.951,A -85,B 0,C 180,E1 -1364.558,E2 -1364.558} C_VEL
LIN {X 0,Y 587.142,Z 186.419,A -85,B 0,C 180,E1 -1367.412,E2 -1367.412} C_VEL
LIN {X 0,Y 587.186,Z 182.269,A -85,B 0,C 180,E1 -1369.581,E2 -1369.581} C_VEL
LIN {X 0,Y 587.188,Z 178.12,A -85,B 0,C 180,E1 -1371.78,E2 -1371.78} C_VEL
LIN {X 0,Y 587.214,Z 173.057,A -85,B 0,C 180,E1 -1374.55,E2 -1374.55} C_VEL
LIN {X 0,Y 587.234,Z 168.648,A -85,B 0,C 180,E1 -1377.051,E2 -1377.051} C_VEL
LIN {X 0,Y 587.257,Z 164.59,A -85,B 0,C 180,E1 -1379.385,E2 -1379.385} C_VEL
LIN {X 0,Y 587.295,Z 160.411,A -85,B 0,C 180,E1 -1381.827,E2 -1381.827} C_VEL
LIN {X 0,Y 587.317,Z 156.179,A -85,B 0,C 180,E1 -1384.343,E2 -1384.343} C_VEL
LIN {X 0,Y 587.258,Z 154.335,A -85,B 0,C 180,E1 -1385.532,E2 -1385.532} C_VEL
LIN {X 0,Y 587.287,Z 154.327,A -85,B 0,C 180,E1 -1387.831,E2 -1387.831} C_VEL
LIN {X 0,Y 587.302,Z 154.331,A -85,B 0,C 180,E1 -1390.255,E2 -1390.255} C_VEL
LIN {X 0,Y 587.315,Z 154.324,A -85,B 0,C 180,E1 -1393.118,E2 -1393.118} C_VEL
LIN {X 0,Y 587.314,Z 154.325,A -85,B 0,C 180,E1 -1396.048,E2 -1396.048} C_VEL
LIN {X 0,Y 587.337,Z 154.328,A -85,B 0,C 180,E1 -1398.925,E2 -1398.925} C_VEL
LIN {X 0,Y 587.311,Z 154.324,A -85,B 0,C 180,E1 -1401.519,E2 -1401.519} C_VEL
LIN {X 0,Y 587.276,Z 154.335,A -85,B 0,C 180,E1 -1404.099,E2 -1404.099} C_VEL
LIN {X 0,Y 587.337,Z 154.321,A -85,B 0,C 180,E1 -1406.889,E2 -1406.889} C_VEL
LIN {X 0,Y 587.335,Z 154.322,A -85,B 0,C 180,E1 -1409.83,E2 -1409.83} C_VEL
LIN {X 0,Y 587.353,Z 154.321,A -85,B 0,C 180,E1 -1412.307,E2 -1412.307} C_VEL
LIN {X 0,Y 587.334,Z 154.327,A -85,B 0,C 180,E1 -1414.483,E2 -1414.483} C_VEL
LIN {X 0,Y 587.309,Z 154.324,A -85,B 0,C 180,E1 -1417.134,E2 -1417.134} C_VEL
LIN {X 0,Y 587.32,Z 154.328,A -85,B 0,C 180,E1 -1419.695,E2 -1419.695} C_VEL
LIN {X 0,Y 587.298,Z 154.326,A -85,B 0,C 180,E1 -1421.872,E2 -1421.872} C_VEL
LIN {X 0,Y 587.324,Z 154.323,A -85,B 0,C 180,E1 -1424.025,E2 -1424.025} C_VEL
LIN {X 0,Y 587.358,Z 154.323,A -85,B 0,C 180,E1 -1426.154,E2 -1426.154} C_VEL
LIN {X 0,Y 587.342,Z 154.32,A -85,B 0,C 180,E1 -1428.962,E2 -1428.962} C_VEL
LIN {X 0,Y 587.317,Z 154.327,A -85,B 0,C 180,E1 -1431.744,E2 -1431.744} C_VEL
LIN {X 0,Y 587.336,Z 154.323,A -85,B 0,C 180,E1 -1434.507,E2 -1434.507} C_VEL
LIN {X 0,Y 587.368,Z 154.318,A -85,B 0,C 180,E1 -1437.257,E2 -1437.257} C_VEL
LIN {X 0,Y 587.384,Z 154.322,A -85,B 0,C 180,E1 -1440,E2 -1440} C_VEL
LIN {X 0,Y 587.37,Z 154.317,A -85,B 0,C 180,E1 -1442.743,E2 -1442.743} C_VEL
LIN {X 0,Y 587.346,Z 154.323,A -85,B 0,C 180,E1 -1445.493,E2 -1445.493} C_VEL
LIN {X 0,Y 587.314,Z 154.326,A -85,B 0,C 180,E1 -1448.256,E2 -1448.256} C_VEL
LIN {X 0,Y 587.35,Z 154.319,A -85,B 0,C 180,E1 -1451.134,E2 -1451.134} C_VEL
LIN {X 0,Y 587.366,Z 154.319,A -85,B 0,C 180,E1 -1454.26,E2 -1454.26} C_VEL
LIN {X 0,Y 587.348,Z 154.324,A -85,B 0,C 180,E1 -1457.406,E2 -1457.406} C_VEL
LIN {X 0,Y 587.324,Z 154.326,A -85,B 0,C 180,E1 -1460.305,E2 -1460.305} C_VEL
LIN {X 0,Y 587.306,Z 154.324,A -85,B 0,C 180,E1 -1463.259,E2 -1463.259} C_VEL
LIN {X 0,Y 587.327,Z 154.326,A -85,B 0,C 180,E1 -1465.517,E2 -1465.517} C_VEL
LIN {X 0,Y 587.34,Z 154.323,A -85,B 0,C 180,E1 -1467.818,E2 -1467.818} C_VEL
LIN {X 0,Y 587.338,Z 154.323,A -85,B 0,C 180,E1 -1470.51,E2 -1470.51} C_VEL
LIN {X 0,Y 587.332,Z 154.321,A -85,B 0,C 180,E1 -1473.397,E2 -1473.397} C_VEL
LIN {X 0,Y 587.278,Z 154.334,A -85,B 0,C 180,E1 -1475.901,E2 -1475.901} C_VEL
LIN {X 0,Y 587.301,Z 154.325,A -85,B 0,C 180,E1 -1478.482,E2 -1478.482} C_VEL
LIN {X 0,Y 587.336,Z 154.329,A -85,B 0,C 180,E1 -1481.157,E2 -1481.157} C_VEL
LIN {X 0,Y 587.313,Z 154.326,A -85,B 0,C 180,E1 -1484.112,E2 -1484.112} C_VEL
LIN {X 0,Y 587.315,Z 154.324,A -85,B 0,C 180,E1 -1486.994,E2 -1486.994} C_VEL
LIN {X 0,Y 587.306,Z 154.332,A -85,B 0,C 180,E1 -1489.745,E2 -1489.745} C_VEL
LIN {X 0,Y 587.311,Z 154.325,A -85,B 0,C 180,E1 -1492.39,E2 -1492.39} C_VEL
LIN {X 0,Y 587.34,Z 154.438,A -85,B 0,C 180,E1 -1493.997,E2 -1493.997} C_VEL
LIN {X 0,Y 587.504,Z 159.169,A -85,B 0,C 180,E1 -1495.789,E2 -1495.789} C_VEL
LIN {X 0,Y 587.475,Z 165.847,A -85,B 0,C 180,E1 -1498.239,E2 -1498.239} C_VEL
LIN {X 0,Y 587.455,Z 173.156,A -85,B 0,C 180,E1 -1500.849,E2 -1500.849} C_VEL
LIN {X 0,Y 587.37,Z 181.706,A -85,B 0,C 180,E1 -1503.817,E2 -1503.817} C_VEL
LIN {X 0,Y 587.343,Z 189.221,A -85,B 0,C 180,E1 -1506.368,E2 -1506.368} C_VEL
LIN {X 0,Y 587.299,Z 198.141,A -85,B 0,C 180,E1 -1509.333,E2 -1509.333} C_VEL
LIN {X 0,Y 587.274,Z 207.03,A -85,B 0,C 180,E1 -1512.232,E2 -1512.232} C_VEL
LIN {X 0,Y 587.216,Z 215.935,A -85,B 0,C 180,E1 -1515.089,E2 -1515.089} C_VEL
LIN {X 0,Y 587.164,Z 224.491,A -85,B 0,C 180,E1 -1517.799,E2 -1517.799} C_VEL
LIN {X 0,Y 587.741,Z 229.223,A -85,B 0,C 180,E1 -1517.899,E2 -1517.899} C_VEL
LIN {X 0,Y 587.672,Z 242.491,A -85,B 0,C 180,E1 -1518.226,E2 -1518.226} C_VEL
LIN {X 0,Y 587.566,Z 254.469,A -85,B 0,C 180,E1 -1518.659,E2 -1518.659} C_VEL
LIN {X 0,Y 587.487,Z 266.206,A -85,B 0,C 180,E1 -1519.227,E2 -1519.227} C_VEL
LIN {X 0,Y 587.446,Z 277.474,A -85,B 0,C 180,E1 -1519.923,E2 -1519.923} C_VEL
LIN {X 0,Y 587.384,Z 287.645,A -85,B 0,C 180,E1 -1520.704,E2 -1520.704} C_VEL
LIN {X 0,Y 587.34,Z 296.786,A -85,B 0,C 180,E1 -1521.571,E2 -1521.571} C_VEL
LIN {X 0,Y 587.259,Z 305.69,A -85,B 0,C 180,E1 -1522.608,E2 -1522.608} C_VEL
LIN {X 0,Y 587.195,Z 312.745,A -85,B 0,C 180,E1 -1523.627,E2 -1523.627} C_VEL
LIN {X 0,Y 587.211,Z 317.68,A -85,B 0,C 180,E1 -1524.506,E2 -1524.506} C_VEL
LIN {X 0,Y 587.188,Z 322.371,A -85,B 0,C 180,E1 -1525.538,E2 -1525.538} C_VEL
LIN {X 0,Y 587.193,Z 325.956,A -85,B 0,C 180,E1 -1526.569,E2 -1526.569} C_VEL
LIN {X 0,Y 587.132,Z 327.808,A -85,B 0,C 180,E1 -1527.255,E2 -1527.255} C_VEL
LIN {X 0,Y 587.141,Z 329.201,A -85,B 0,C 180,E1 -1527.942,E2 -1527.942} C_VEL
LIN {X 0,Y 587.14,Z 330.784,A -85,B 0,C 180,E1 -1529.314,E2 -1529.314} C_VEL
LIN {X 0,Y 587.137,Z 331,A -85,B 0,C 180,E1 -1530,E2 -1530} C_VEL
LIN {X 0,Y 587.147,Z 330.185,A -85,B 0,C 180,E1 -1531.372,E2 -1531.372} C_VEL
LIN {X 0,Y 587.141,Z 329.202,A -85,B 0,C 180,E1 -1532.058,E2 -1532.058} C_VEL
LIN {X 0,Y 587.132,Z 327.81,A -85,B 0,C 180,E1 -1532.744,E2 -1532.744} C_VEL
LIN {X 0,Y 587.213,Z 324.897,A -85,B 0,C 180,E1 -1533.774,E2 -1533.774} C_VEL
LIN {X 0,Y 587.147,Z 320.95,A -85,B 0,C 180,E1 -1534.806,E2 -1534.806} C_VEL
LIN {X 0,Y 587.218,Z 314.878,A -85,B 0,C 180,E1 -1536.011,E2 -1536.011} C_VEL
LIN {X 0,Y 587.245,Z 308.237,A -85,B 0,C 180,E1 -1537.046,E2 -1537.046} C_VEL
LIN {X 0,Y 587.299,Z 299.991,A -85,B 0,C 180,E1 -1538.083,E2 -1538.083} C_VEL
LIN {X 0,Y 587.343,Z 291.539,A -85,B 0,C 180,E1 -1538.949,E2 -1538.949} C_VEL
LIN {X 0,Y 587.418,Z 281.095,A -85,B 0,C 180,E1 -1539.816,E2 -1539.816} C_VEL
LIN {X 0,Y 587.447,Z 270.761,A -85,B 0,C 180,E1 -1540.512,E2 -1540.512} C_VEL
LIN {X 0,Y 587.528,Z 259.179,A -85,B 0,C 180,E1 -1541.133,E2 -1541.133} C_VEL
LIN {X 0,Y 587.593,Z 246.706,A -85,B 0,C 180,E1 -1541.636,E2 -1541.636} C_VEL
LIN {X 0,Y 587.74,Z 233.446,A -85,B 0,C 180,E1 -1542.013,E2 -1542.013} C_VEL
LIN {X 0,Y 587.522,Z 226.662,A -85,B 0,C 180,E1 -1542.154,E2 -1542.154} C_VEL
LIN {X 0,Y 587.164,Z 224.492,A -85,B 0,C 180,E1 -1542.2,E2 -1542.2} C_VEL
LIN {X 0,Y 587.215,Z 215.936,A -85,B 0,C 180,E1 -1544.911,E2 -1544.911} C_VEL
LIN {X 0,Y 587.274,Z 207.031,A -85,B 0,C 180,E1 -1547.768,E2 -1547.768} C_VEL
LIN {X 0,Y 587.298,Z 198.142,A -85,B 0,C 180,E1 -1550.667,E2 -1550.667} C_VEL
LIN {X 0,Y 587.343,Z 189.222,A -85,B 0,C 180,E1 -1553.631,E2 -1553.631} C_VEL
LIN {X 0,Y 587.37,Z 181.431,A -85,B 0,C 180,E1 -1556.277,E2 -1556.277} C_VEL
LIN {X 0,Y 587.454,Z 173.156,A -85,B 0,C 180,E1 -1559.151,E2 -1559.151} C_VEL
LIN {X 0,Y 587.468,Z 165.59,A -85,B 0,C 180,E1 -1561.855,E2 -1561.855} C_VEL
LIN {X 0,Y 587.527,Z 158.73,A -85,B 0,C 180,E1 -1564.373,E2 -1564.373} C_VEL
LIN {X 0,Y 587.308,Z 154.33,A -85,B 0,C 180,E1 -1566.057,E2 -1566.057} C_VEL
LIN {X 0,Y 587.305,Z 154.328,A -85,B 0,C 180,E1 -1568.938,E2 -1568.938} C_VEL
LIN {X 0,Y 587.33,Z 154.322,A -85,B 0,C 180,E1 -1571.157,E2 -1571.157} C_VEL
LIN {X 0,Y 587.326,Z 154.325,A -85,B 0,C 180,E1 -1574.113,E2 -1574.113} C_VEL
LIN {X 0,Y 587.312,Z 154.329,A -85,B 0,C 180,E1 -1576.993,E2 -1576.993} C_VEL
LIN {X 0,Y 587.304,Z 154.325,A -85,B 0,C 180,E1 -1579.745,E2 -1579.745} C_VEL
LIN {X 0,Y 587.312,Z 154.33,A -85,B 0,C 180,E1 -1582.39,E2 -1582.39} C_VEL
LIN {X 0,Y 587.338,Z 154.327,A -85,B 0,C 180,E1 -1585.653,E2 -1585.653} C_VEL
LIN {X 0,Y 587.342,Z 154.32,A -85,B 0,C 180,E1 -1588.231,E2 -1588.231} C_VEL
LIN {X 0,Y 587.348,Z 154.326,A -85,B 0,C 180,E1 -1590.866,E2 -1590.866} C_VEL
LIN {X 0,Y 587.359,Z 154.32,A -85,B 0,C 180,E1 -1593.818,E2 -1593.818} C_VEL
LIN {X 0,Y 587.323,Z 154.33,A -85,B 0,C 180,E1 -1595.993,E2 -1595.993} C_VEL
LIN {X 0,Y 587.329,Z 154.323,A -85,B 0,C 180,E1 -1598.962,E2 -1598.962} C_VEL
LIN {X 0,Y 587.305,Z 154.325,A -85,B 0,C 180,E1 -1601.873,E2 -1601.873} C_VEL
LIN {X 0,Y 587.323,Z 154.324,A -85,B 0,C 180,E1 -1604.025,E2 -1604.025} C_VEL
LIN {X 0,Y 587.356,Z 154.325,A -85,B 0,C 180,E1 -1606.154,E2 -1606.154} C_VEL
LIN {X 0,Y 587.34,Z 154.32,A -85,B 0,C 180,E1 -1608.962,E2 -1608.962} C_VEL
LIN {X 0,Y 587.314,Z 154.326,A -85,B 0,C 180,E1 -1611.744,E2 -1611.744} C_VEL
LIN {X 0,Y 587.342,Z 154.323,A -85,B 0,C 180,E1 -1614.507,E2 -1614.507} C_VEL
LIN {X 0,Y 587.369,Z 154.317,A -85,B 0,C 180,E1 -1617.257,E2 -1617.257} C_VEL
LIN {X 0,Y 587.383,Z 154.322,A -85,B 0,C 180,E1 -1620,E2 -1620} C_VEL
LIN {X 0,Y 587.368,Z 154.317,A -85,B 0,C 180,E1 -1622.743,E2 -1622.743} C_VEL
LIN {X 0,Y 587.34,Z 154.323,A -85,B 0,C 180,E1 -1625.493,E2 -1625.493} C_VEL
LIN {X 0,Y 587.314,Z 154.327,A -85,B 0,C 180,E1 -1628.256,E2 -1628.256} C_VEL
LIN {X 0,Y 587.346,Z 154.319,A -85,B 0,C 180,E1 -1631.134,E2 -1631.134} C_VEL
LIN {X 0,Y 587.364,Z 154.318,A -85,B 0,C 180,E1 -1634.261,E2 -1634.261} C_VEL
LIN {X 0,Y 587.347,Z 154.323,A -85,B 0,C 180,E1 -1637.406,E2 -1637.406} C_VEL
LIN {X 0,Y 587.306,Z 154.326,A -85,B 0,C 180,E1 -1638.3,E2 -1638.3} C_VEL
LIN {X 0,Y 586.666,Z 154.411,A -85,B 0,C 180,E1 -1638.872,E2 -1638.872} C_VEL
LIN {X 0,Y 583.848,Z 154.759,A -85,B 0,C 180,E1 -1639.8,E2 -1639.8} C_VEL
LIN {X 0,Y 581.438,Z 155.063,A -85,B 0,C 180,E1 -1640.547,E2 -1640.547} C_VEL
LIN {X 0,Y 580.377,Z 155.189,A -85,B 0,C 180,E1 -1641.123,E2 -1641.123} C_VEL
LIN {X 0,Y 580.278,Z 155.2,A -85,B 0,C 180,E1 -1641.319,E2 -1641.319} C_VEL
LIN {X 0,Y 580.294,Z 155.2,A -85,B 0,C 180,E1 -1644.317,E2 -1644.317} C_VEL
LIN {X 0,Y 580.275,Z 155.2,A -85,B 0,C 180,E1 -1646.624,E2 -1646.624} C_VEL
LIN {X 0,Y 580.3,Z 155.202,A -85,B 0,C 180,E1 -1649.31,E2 -1649.31} C_VEL
LIN {X 0,Y 580.298,Z 155.201,A -85,B 0,C 180,E1 -1652.201,E2 -1652.201} C_VEL
LIN {X 0,Y 580.277,Z 155.202,A -85,B 0,C 180,E1 -1654.697,E2 -1654.697} C_VEL
LIN {X 0,Y 580.267,Z 155.204,A -85,B 0,C 180,E1 -1657.271,E2 -1657.271} C_VEL
LIN {X 0,Y 580.286,Z 155.199,A -85,B 0,C 180,E1 -1660.27,E2 -1660.27} C_VEL
LIN {X 0,Y 580.276,Z 155.206,A -85,B 0,C 180,E1 -1662.707,E2 -1662.707} C_VEL
LIN {X 0,Y 580.27,Z 155.202,A -85,B 0,C 180,E1 -1665.609,E2 -1665.609} C_VEL
LIN {X 0,Y 580.279,Z 155.204,A -85,B 0,C 180,E1 -1668.232,E2 -1668.232} C_VEL
LIN {X 0,Y 580.261,Z 155.205,A -85,B 0,C 180,E1 -1670.964,E2 -1670.964} C_VEL
LIN {X 0,Y 580.24,Z 155.207,A -85,B 0,C 180,E1 -1673.595,E2 -1673.595} C_VEL
LIN {X 0,Y 580.213,Z 155.211,A -85,B 0,C 180,E1 -1674.45,E2 -1674.45} C_VEL
LIN {X 0,Y 580.206,Z 157.693,A -85,B 0,C 180,E1 -1676.138,E2 -1676.138} C_VEL
LIN {X 0,Y 580.215,Z 161.826,A -85,B 0,C 180,E1 -1678.611,E2 -1678.611} C_VEL
LIN {X 0,Y 580.226,Z 165.873,A -85,B 0,C 180,E1 -1681.021,E2 -1681.021} C_VEL
LIN {X 0,Y 580.2,Z 170.462,A -85,B 0,C 180,E1 -1683.685,E2 -1683.685} C_VEL
LIN {X 0,Y 580.136,Z 175.303,A -85,B 0,C 180,E1 -1686.436,E2 -1686.436} C_VEL
LIN {X 0,Y 580.132,Z 179.688,A -85,B 0,C 180,E1 -1688.879,E2 -1688.879} C_VEL
LIN {X 0,Y 580.092,Z 184.865,A -85,B 0,C 180,E1 -1691.64,E2 -1691.64} C_VEL
LIN {X 0,Y 580.071,Z 190.395,A -85,B 0,C 180,E1 -1694.541,E2 -1694.541} C_VEL
LIN {X 0,Y 580.059,Z 195.924,A -85,B 0,C 180,E1 -1697.403,E2 -1697.403} C_VEL
LIN {X 0,Y 580.067,Z 196.529,A -85,B 0,C 180,E1 -1697.715,E2 -1697.715} C_VEL
LIN {X 0,Y 580.786,Z 202.5,A -85,B 0,C 180,E1 -1697.863,E2 -1697.863} C_VEL
LIN {X 0,Y 580.669,Z 215.159,A -85,B 0,C 180,E1 -1698.215,E2 -1698.215} C_VEL
LIN {X 0,Y 580.578,Z 226.885,A -85,B 0,C 180,E1 -1698.673,E2 -1698.673} C_VEL
LIN {X 0,Y 580.505,Z 238.554,A -85,B 0,C 180,E1 -1699.273,E2 -1699.273} C_VEL
LIN {X 0,Y 580.439,Z 249.329,A -85,B 0,C 180,E1 -1699.977,E2 -1699.977} C_VEL
LIN {X 0,Y 580.333,Z 259.105,A -85,B 0,C 180,E1 -1700.767,E2 -1700.767} C_VEL
LIN {X 0,Y 580.264,Z 267.998,A -85,B 0,C 180,E1 -1701.643,E2 -1701.643} C_VEL
LIN {X 0,Y 580.205,Z 276.682,A -85,B 0,C 180,E1 -1702.693,E2 -1702.693} C_VEL
LIN {X 0,Y 580.137,Z 283.609,A -85,B 0,C 180,E1 -1703.741,E2 -1703.741} C_VEL
LIN {X 0,Y 580.086,Z 289.158,A -85,B 0,C 180,E1 -1704.787,E2 -1704.787} C_VEL
LIN {X 0,Y 580.105,Z 293.518,A -85,B 0,C 180,E1 -1705.832,E2 -1705.832} C_VEL
LIN {X 0,Y 580.123,Z 295.822,A -85,B 0,C 180,E1 -1706.527,E2 -1706.527} C_VEL
LIN {X 0,Y 580.043,Z 297.699,A -85,B 0,C 180,E1 -1707.222,E2 -1707.222} C_VEL
LIN {X 0,Y 580.04,Z 299.127,A -85,B 0,C 180,E1 -1707.917,E2 -1707.917} C_VEL
LIN {X 0,Y 580.04,Z 300.755,A -85,B 0,C 180,E1 -1709.306,E2 -1709.306} C_VEL
LIN {X 0,Y 580.038,Z 300.996,A -85,B 0,C 180,E1 -1710,E2 -1710} C_VEL
LIN {X 0,Y 580.04,Z 300.815,A -85,B 0,C 180,E1 -1710.694,E2 -1710.694} C_VEL
LIN {X 0,Y 580.04,Z 299.271,A -85,B 0,C 180,E1 -1712.083,E2 -1712.083} C_VEL
LIN {X 0,Y 580.044,Z 297.91,A -85,B 0,C 180,E1 -1712.778,E2 -1712.778} C_VEL
LIN {X 0,Y 580.11,Z 295.033,A -85,B 0,C 180,E1 -1713.821,E2 -1713.821} C_VEL
LIN {X 0,Y 580.053,Z 291.133,A -85,B 0,C 180,E1 -1714.865,E2 -1714.865} C_VEL
LIN {X 0,Y 580.162,Z 286.101,A -85,B 0,C 180,E1 -1715.91,E2 -1715.91} C_VEL
LIN {X 0,Y 580.158,Z 279.779,A -85,B 0,C 180,E1 -1716.958,E2 -1716.958} C_VEL
LIN {X 0,Y 580.241,Z 271.859,A -85,B 0,C 180,E1 -1718.007,E2 -1718.007} C_VEL
LIN {X 0,Y 580.308,Z 262.009,A -85,B 0,C 180,E1 -1719.058,E2 -1719.058} C_VEL
LIN {X 0,Y 580.406,Z 251.69,A -85,B 0,C 180,E1 -1719.936,E2 -1719.936} C_VEL
LIN {X 0,Y 580.474,Z 240.053,A -85,B 0,C 180,E1 -1720.728,E2 -1720.728} C_VEL
LIN {X 0,Y 580.548,Z 229.209,A -85,B 0,C 180,E1 -1721.312,E2 -1721.312} C_VEL
LIN {X 0,Y 580.671,Z 216.621,A -85,B 0,C 180,E1 -1721.825,E2 -1721.825} C_VEL
LIN {X 0,Y 580.77,Z 203.46,A -85,B 0,C 180,E1 -1722.204,E2 -1722.204} C_VEL
LIN {X 0,Y 580.465,Z 199.254,A -85,B 0,C 180,E1 -1722.299,E2 -1722.299} C_VEL
LIN {X 0,Y 580.079,Z 196.531,A -85,B 0,C 180,E1 -1722.374,E2 -1722.374} C_VEL
LIN {X 0,Y 580.057,Z 191.95,A -85,B 0,C 180,E1 -1724.74,E2 -1724.74} C_VEL
LIN {X 0,Y 580.068,Z 187.801,A -85,B 0,C 180,E1 -1726.905,E2 -1726.905} C_VEL
LIN {X 0,Y 580.098,Z 182.268,A -85,B 0,C 180,E1 -1729.83,E2 -1729.83} C_VEL
LIN {X 0,Y 580.127,Z 178.145,A -85,B 0,C 180,E1 -1732.059,E2 -1732.059} C_VEL
LIN {X 0,Y 580.159,Z 172.782,A -85,B 0,C 180,E1 -1735.087,E2 -1735.087} C_VEL
LIN {X 0,Y 580.222,Z 167.993,A -85,B 0,C 180,E1 -1737.844,E2 -1737.844} C_VEL
LIN {X 0,Y 580.201,Z 163.163,A -85,B 0,C 180,E1 -1740.68,E2 -1740.68} C_VEL
LIN {X 0,Y 580.238,Z 158.765,A -85,B 0,C 180,E1 -1743.306,E2 -1743.306} C_VEL
LIN {X 0,Y 580.216,Z 155.212,A -85,B 0,C 180,E1 -1745.55,E2 -1745.55} C_VEL
LIN {X 0,Y 580.243,Z 155.206,A -85,B 0,C 180,E1 -1748.15,E2 -1748.15} C_VEL
LIN {X 0,Y 580.279,Z 155.202,A -85,B 0,C 180,E1 -1750.845,E2 -1750.845} C_VEL
LIN {X 0,Y 580.28,Z 155.205,A -85,B 0,C 180,E1 -1753.658,E2 -1753.658} C_VEL
LIN {X 0,Y 580.275,Z 155.201,A -85,B 0,C 180,E1 -1756.61,E2 -1756.61} C_VEL
LIN {X 0,Y 580.298,Z 155.202,A -85,B 0,C 180,E1 -1759.156,E2 -1759.156} C_VEL
LIN {X 0,Y 580.278,Z 155.202,A -85,B 0,C 180,E1 -1761.929,E2 -1761.929} C_VEL
LIN {X 0,Y 580.227,Z 155.21,A -85,B 0,C 180,E1 -1764.451,E2 -1764.451} C_VEL
LIN {X 0,Y 580.289,Z 155.2,A -85,B 0,C 180,E1 -1766.975,E2 -1766.975} C_VEL
LIN {X 0,Y 580.297,Z 155.203,A -85,B 0,C 180,E1 -1769.425,E2 -1769.425} C_VEL
LIN {X 0,Y 580.299,Z 155.199,A -85,B 0,C 180,E1 -1772.141,E2 -1772.141} C_VEL
LIN {X 0,Y 580.322,Z 155.194,A -85,B 0,C 180,E1 -1775.27,E2 -1775.27} C_VEL
LIN {X 0,Y 580.251,Z 155.209,A -85,B 0,C 180,E1 -1777.946,E2 -1777.946} C_VEL
LIN {X 0,Y 580.298,Z 155.2,A -85,B 0,C 180,E1 -1780.849,E2 -1780.849} C_VEL
LIN {X 0,Y 580.279,Z 155.2,A -85,B 0,C 180,E1 -1783.825,E2 -1783.825} C_VEL
LIN {X 0,Y 580.326,Z 155.197,A -85,B 0,C 180,E1 -1785.983,E2 -1785.983} C_VEL
LIN {X 0,Y 580.306,Z 155.197,A -85,B 0,C 180,E1 -1788.827,E2 -1788.827} C_VEL
LIN {X 0,Y 580.291,Z 155.204,A -85,B 0,C 180,E1 -1791.643,E2 -1791.643} C_VEL
LIN {X 0,Y 580.301,Z 155.199,A -85,B 0,C 180,E1 -1794.44,E2 -1794.44} C_VEL
LIN {X 0,Y 580.335,Z 155.194,A -85,B 0,C 180,E1 -1797.223,E2 -1797.223} C_VEL
LIN {X 0,Y 580.353,Z 155.198,A -85,B 0,C 180,E1 -1800,E2 -1800} C_VEL
LIN {X 0,Y 580.337,Z 155.193,A -85,B 0,C 180,E1 -1802.777,E2 -1802.777} C_VEL
LIN {X 0,Y 580.31,Z 155.198,A -85,B 0,C 180,E1 -1805.56,E2 -1805.56} C_VEL
LIN {X 0,Y 580.289,Z 155.202,A -85,B 0,C 180,E1 -1808.357,E2 -1808.357} C_VEL
LIN {X 0,Y 580.301,Z 155.197,A -85,B 0,C 180,E1 -1811.191,E2 -1811.191} C_VEL
LIN {X 0,Y 580.326,Z 155.198,A -85,B 0,C 180,E1 -1814.017,E2 -1814.017} C_VEL
LIN {X 0,Y 580.314,Z 155.2,A -85,B 0,C 180,E1 -1816.914,E2 -1816.914} C_VEL
LIN {X 0,Y 580.284,Z 155.199,A -85,B 0,C 180,E1 -1819.823,E2 -1819.823} C_VEL
LIN {X 0,Y 580.26,Z 155.206,A -85,B 0,C 180,E1 -1822.053,E2 -1822.053} C_VEL
LIN {X 0,Y 580.303,Z 155.197,A -85,B 0,C 180,E1 -1825.08,E2 -1825.08} C_VEL
LIN {X 0,Y 580.295,Z 155.198,A -85,B 0,C 180,E1 -1828.186,E2 -1828.186} C_VEL
LIN {X 0,Y 580.286,Z 155.204,A -85,B 0,C 180,E1 -1830.695,E2 -1830.695} C_VEL
LIN {X 0,Y 580.302,Z 155.197,A -85,B 0,C 180,E1 -1833.316,E2 -1833.316} C_VEL
LIN {X 0,Y 580.229,Z 155.21,A -85,B 0,C 180,E1 -1835.754,E2 -1835.754} C_VEL
LIN {X 0,Y 580.271,Z 155.203,A -85,B 0,C 180,E1 -1838.148,E2 -1838.148} C_VEL
LIN {X 0,Y 580.296,Z 155.201,A -85,B 0,C 180,E1 -1840.844,E2 -1840.844} C_VEL
LIN {X 0,Y 580.274,Z 155.201,A -85,B 0,C 180,E1 -1843.659,E2 -1843.659} C_VEL
LIN {X 0,Y 580.275,Z 155.203,A -85,B 0,C 180,E1 -1846.61,E2 -1846.61} C_VEL
LIN {X 0,Y 580.294,Z 155.199,A -85,B 0,C 180,E1 -1849.156,E2 -1849.156} C_VEL
LIN {X 0,Y 580.276,Z 155.203,A -85,B 0,C 180,E1 -1851.929,E2 -1851.929} C_VEL
LIN {X 0,Y 580.306,Z 155.379,A -85,B 0,C 180,E1 -1853.855,E2 -1853.855} C_VEL
LIN {X 0,Y 580.535,Z 159.169,A -85,B 0,C 180,E1 -1855.32,E2 -1855.32} C_VEL
LIN {X 0,Y 580.479,Z 166.204,A -85,B 0,C 180,E1 -1857.942,E2 -1857.942} C_VEL
LIN {X 0,Y 580.461,Z 173.714,A -85,B 0,C 180,E1 -1860.663,E2 -1860.663} C_VEL
LIN {X 0,Y 580.354,Z 182.216,A -85,B 0,C 180,E1 -1863.654,E2 -1863.654} C_VEL
LIN {X 0,Y 580.3,Z 190.334,A -85,B 0,C 180,E1 -1866.443,E2 -1866.443} C_VEL
LIN {X 0,Y 580.241,Z 199.239,A -85,B 0,C 180,E1 -1869.436,E2 -1869.436} C_VEL
LIN {X 0,Y 580.201,Z 208.143,A -85,B 0,C 180,E1 -1872.372,E2 -1872.372} C_VEL
LIN {X 0,Y 580.141,Z 217.048,A -85,B 0,C 180,E1 -1875.262,E2 -1875.262} C_VEL
LIN {X 0,Y 580.097,Z 224.491,A -85,B 0,C 180,E1 -1877.648,E2 -1877.648} C_VEL
LIN {X 0,Y 580.801,Z 230.365,A -85,B 0,C 180,E1 -1877.774,E2 -1877.774} C_VEL
LIN {X 0,Y 580.722,Z 242.492,A -85,B 0,C 180,E1 -1878.083,E2 -1878.083} C_VEL
LIN {X 0,Y 580.594,Z 254.318,A -85,B 0,C 180,E1 -1878.514,E2 -1878.514} C_VEL
LIN {X 0,Y 580.501,Z 266.207,A -85,B 0,C 180,E1 -1879.096,E2 -1879.096} C_VEL
LIN {X 0,Y 580.441,Z 277.475,A -85,B 0,C 180,E1 -1879.8,E2 -1879.8} C_VEL
LIN {X 0,Y 580.352,Z 287.645,A -85,B 0,C 180,E1 -1880.591,E2 -1880.591} C_VEL
LIN {X 0,Y 580.279,Z 296.786,A -85,B 0,C 180,E1 -1881.468,E2 -1881.468} C_VEL
LIN {X 0,Y 580.199,Z 305.69,A -85,B 0,C 180,E1 -1882.518,E2 -1882.518} C_VEL
LIN {X 0,Y 580.12,Z 312.465,A -85,B 0,C 180,E1 -1883.505,E2 -1883.505} C_VEL
LIN {X 0,Y 580.139,Z 317.68,A -85,B 0,C 180,E1 -1884.438,E2 -1884.438} C_VEL
LIN {X 0,Y 580.108,Z 322.371,A -85,B 0,C 180,E1 -1885.483,E2 -1885.483} C_VEL
LIN {X 0,Y 580.123,Z 325.956,A -85,B 0,C 180,E1 -1886.527,E2 -1886.527} C_VEL
LIN {X 0,Y 580.043,Z 327.808,A -85,B 0,C 180,E1 -1887.222,E2 -1887.222} C_VEL
LIN {X 0,Y 580.04,Z 329.201,A -85,B 0,C 180,E1 -1887.917,E2 -1887.917} C_VEL
LIN {X 0,Y 580.04,Z 330.784,A -85,B 0,C 180,E1 -1889.306,E2 -1889.306} C_VEL
LIN {X 0,Y 580.037,Z 331,A -85,B 0,C 180,E1 -1890,E2 -1890} C_VEL
LIN {X 0,Y 580.047,Z 330.185,A -85,B 0,C 180,E1 -1891.388,E2 -1891.388} C_VEL
LIN {X 0,Y 580.04,Z 329.202,A -85,B 0,C 180,E1 -1892.083,E2 -1892.083} C_VEL
LIN {X 0,Y 580.043,Z 327.81,A -85,B 0,C 180,E1 -1892.778,E2 -1892.778} C_VEL
LIN {X 0,Y 580.11,Z 324.897,A -85,B 0,C 180,E1 -1893.82,E2 -1893.82} C_VEL
LIN {X 0,Y 580.053,Z 320.95,A -85,B 0,C 180,E1 -1894.865,E2 -1894.865} C_VEL
LIN {X 0,Y 580.139,Z 314.879,A -85,B 0,C 180,E1 -1896.085,E2 -1896.085} C_VEL
LIN {X 0,Y 580.184,Z 308.237,A -85,B 0,C 180,E1 -1897.132,E2 -1897.132} C_VEL
LIN {X 0,Y 580.25,Z 299.991,A -85,B 0,C 180,E1 -1898.182,E2 -1898.182} C_VEL
LIN {X 0,Y 580.308,Z 291.539,A -85,B 0,C 180,E1 -1899.058,E2 -1899.058} C_VEL
LIN {X 0,Y 580.412,Z 281.096,A -85,B 0,C 180,E1 -1899.936,E2 -1899.936} C_VEL
LIN {X 0,Y 580.451,Z 270.762,A -85,B 0,C 180,E1 -1900.64,E2 -1900.64} C_VEL
LIN {X 0,Y 580.563,Z 259.598,A -85,B 0,C 180,E1 -1901.247,E2 -1901.247} C_VEL
LIN {X 0,Y 580.636,Z 247.773,A -85,B 0,C 180,E1 -1901.741,E2 -1901.741} C_VEL
LIN {X 0,Y 580.773,Z 234.36,A -85,B 0,C 180,E1 -1902.137,E2 -1902.137} C_VEL
LIN {X 0,Y 580.672,Z 228.099,A -85,B 0,C 180,E1 -1902.272,E2 -1902.272} C_VEL
LIN {X 0,Y 580.097,Z 224.492,A -85,B 0,C 180,E1 -1902.351,E2 -1902.351} C_VEL
LIN {X 0,Y 580.153,Z 215.936,A -85,B 0,C 180,E1 -1905.097,E2 -1905.097} C_VEL
LIN {X 0,Y 580.199,Z 207.031,A -85,B 0,C 180,E1 -1907.992,E2 -1907.992} C_VEL
LIN {X 0,Y 580.241,Z 199.24,A -85,B 0,C 180,E1 -1910.564,E2 -1910.564} C_VEL
LIN {X 0,Y 580.3,Z 190.336,A -85,B 0,C 180,E1 -1913.557,E2 -1913.557} C_VEL
LIN {X 0,Y 580.353,Z 182.217,A -85,B 0,C 180,E1 -1916.346,E2 -1916.346} C_VEL
LIN {X 0,Y 580.46,Z 173.715,A -85,B 0,C 180,E1 -1919.337,E2 -1919.337} C_VEL
LIN {X 0,Y 580.478,Z 165.848,A -85,B 0,C 180,E1 -1922.189,E2 -1922.189} C_VEL
LIN {X 0,Y 580.535,Z 159.17,A -85,B 0,C 180,E1 -1924.679,E2 -1924.679} C_VEL
LIN {X 0,Y 580.283,Z 155.215,A -85,B 0,C 180,E1 -1926.21,E2 -1926.21} C_VEL
LIN {X 0,Y 580.281,Z 155.201,A -85,B 0,C 180,E1 -1929.183,E2 -1929.183} C_VEL
LIN {X 0,Y 580.288,Z 155.204,A -85,B 0,C 180,E1 -1931.768,E2 -1931.768} C_VEL
LIN {X 0,Y 580.26,Z 155.203,A -85,B 0,C 180,E1 -1934.626,E2 -1934.626} C_VEL
LIN {X 0,Y 580.285,Z 155.201,A -85,B 0,C 180,E1 -1937.628,E2 -1937.628} C_VEL
LIN {X 0,Y 580.277,Z 155.201,A -85,B 0,C 180,E1 -1940.066,E2 -1940.066} C_VEL
LIN {X 0,Y 580.262,Z 155.202,A -85,B 0,C 180,E1 -1943.07,E2 -1943.07} C_VEL
LIN {X 0,Y 580.31,Z 155.198,A -85,B 0,C 180,E1 -1946.145,E2 -1946.145} C_VEL
LIN {X 0,Y 580.278,Z 155.202,A -85,B 0,C 180,E1 -1948.615,E2 -1948.615} C_VEL
LIN {X 0,Y 580.29,Z 155.204,A -85,B 0,C 180,E1 -1951.024,E2 -1951.024} C_VEL
LIN {X 0,Y 580.29,Z 155.199,A -85,B 0,C 180,E1 -1953.666,E2 -1953.666} C_VEL
LIN {X 0,Y 580.294,Z 155.201,A -85,B 0,C 180,E1 -1955.683,E2 -1955.683} C_VEL
LIN {X 0,Y 580.28,Z 155.2,A -85,B 0,C 180,E1 -1958.694,E2 -1958.694} C_VEL
LIN {X 0,Y 580.297,Z 155.202,A -85,B 0,C 180,E1 -1960.913,E2 -1960.913} C_VEL
LIN {X 0,Y 580.278,Z 155.201,A -85,B 0,C 180,E1 -1963.826,E2 -1963.826} C_VEL
LIN {X 0,Y 580.323,Z 155.198,A -85,B 0,C 180,E1 -1965.983,E2 -1965.983} C_VEL
LIN {X 0,Y 580.303,Z 155.197,A -85,B 0,C 180,E1 -1968.827,E2 -1968.827} C_VEL
LIN {X 0,Y 580.288,Z 155.203,A -85,B 0,C 180,E1 -1971.643,E2 -1971.643} C_VEL
LIN {X 0,Y 580.306,Z 155.198,A -85,B 0,C 180,E1 -1974.44,E2 -1974.44} C_VEL
LIN {X 0,Y 580.336,Z 155.193,A -85,B 0,C 180,E1 -1977.223,E2 -1977.223} C_VEL
LIN {X 0,Y 580.352,Z 155.198,A -85,B 0,C 180,E1 -1980,E2 -1980} C_VEL
LIN {X 0,Y 580.335,Z 155.194,A -85,B 0,C 180,E1 -1982.777,E2 -1982.777} C_VEL
LIN {X 0,Y 580.304,Z 155.199,A -85,B 0,C 180,E1 -1985.56,E2 -1985.56} C_VEL
LIN {X 0,Y 580.289,Z 155.203,A -85,B 0,C 180,E1 -1988.357,E2 -1988.357} C_VEL
LIN {X 0,Y 580.298,Z 155.197,A -85,B 0,C 180,E1 -1991.191,E2 -1991.191} C_VEL
LIN {X 0,Y 580.324,Z 155.198,A -85,B 0,C 180,E1 -1994.017,E2 -1994.017} C_VEL
LIN {X 0,Y 580.311,Z 155.201,A -85,B 0,C 180,E1 -1996.914,E2 -1996.914} C_VEL
LIN {X 0,Y 580.281,Z 155.2,A -85,B 0,C 180,E1 -1999.823,E2 -1999.823} C_VEL
LIN {X 0,Y 580.278,Z 155.2,A -85,B 0,C 180,E1 -2001.319,E2 -2001.319} C_VEL
LIN {X 0,Y 579.57,Z 155.292,A -85,B 0,C 180,E1 -2001.898,E2 -2001.898} C_VEL
LIN {X 0,Y 576.691,Z 155.649,A -85,B 0,C 180,E1 -2002.838,E2 -2002.838} C_VEL
LIN {X 0,Y 574.303,Z 155.947,A -85,B 0,C 180,E1 -2003.594,E2 -2003.594} C_VEL
LIN {X 0,Y 573.309,Z 156.072,A -85,B 0,C 180,E1 -2004.178,E2 -2004.178} C_VEL
LIN {X 0,Y 573.243,Z 156.077,A -85,B 0,C 180,E1 -2004.375,E2 -2004.375} C_VEL
LIN {X 0,Y 573.249,Z 156.078,A -85,B 0,C 180,E1 -2006.976,E2 -2006.976} C_VEL
LIN {X 0,Y 573.246,Z 156.079,A -85,B 0,C 180,E1 -2009.489,E2 -2009.489} C_VEL
LIN {X 0,Y 573.253,Z 156.082,A -85,B 0,C 180,E1 -2012.645,E2 -2012.645} C_VEL
LIN {X 0,Y 573.19,Z 156.084,A -85,B 0,C 180,E1 -2015.189,E2 -2015.189} C_VEL
LIN {X 0,Y 573.216,Z 156.085,A -85,B 0,C 180,E1 -2017.809,E2 -2017.809} C_VEL
LIN {X 0,Y 573.244,Z 156.077,A -85,B 0,C 180,E1 -2020.525,E2 -2020.525} C_VEL
LIN {X 0,Y 573.236,Z 156.078,A -85,B 0,C 180,E1 -2023.36,E2 -2023.36} C_VEL
LIN {X 0,Y 573.244,Z 156.083,A -85,B 0,C 180,E1 -2026.331,E2 -2026.331} C_VEL
LIN {X 0,Y 573.226,Z 156.08,A -85,B 0,C 180,E1 -2028.543,E2 -2028.543} C_VEL
LIN {X 0,Y 573.228,Z 156.085,A -85,B 0,C 180,E1 -2031.298,E2 -2031.298} C_VEL
LIN {X 0,Y 573.181,Z 156.085,A -85,B 0,C 180,E1 -2034.023,E2 -2034.023} C_VEL
LIN {X 0,Y 573.165,Z 156.362,A -85,B 0,C 180,E1 -2034.81,E2 -2034.81} C_VEL
LIN {X 0,Y 573.18,Z 161.266,A -85,B 0,C 180,E1 -2037.784,E2 -2037.784} C_VEL
LIN {X 0,Y 573.149,Z 165.986,A -85,B 0,C 180,E1 -2040.628,E2 -2040.628} C_VEL
LIN {X 0,Y 573.124,Z 170.029,A -85,B 0,C 180,E1 -2043.018,E2 -2043.018} C_VEL
LIN {X 0,Y 573.105,Z 174.081,A -85,B 0,C 180,E1 -2045.359,E2 -2045.359} C_VEL
LIN {X 0,Y 573.05,Z 178.105,A -85,B 0,C 180,E1 -2047.655,E2 -2047.655} C_VEL
LIN {X 0,Y 573.016,Z 182.135,A -85,B 0,C 180,E1 -2049.915,E2 -2049.915} C_VEL
LIN {X 0,Y 572.97,Z 186.248,A -85,B 0,C 180,E1 -2052.143,E2 -2052.143} C_VEL
LIN {X 0,Y 572.98,Z 191.778,A -85,B 0,C 180,E1 -2055.074,E2 -2055.074} C_VEL
LIN {X 0,Y 572.979,Z 196.53,A -85,B 0,C 180,E1 -2057.56,E2 -2057.56} C_VEL
LIN {X 0,Y 573.854,Z 203.437,A -85,B 0,C 180,E1 -2057.737,E2 -2057.737} C_VEL
LIN {X 0,Y 573.709,Z 216.474,A -85,B 0,C 180,E1 -2058.115,E2 -2058.115} C_VEL
LIN {X 0,Y 573.584,Z 228.667,A -85,B 0,C 180,E1 -2058.614,E2 -2058.614} C_VEL
LIN {X 0,Y 573.508,Z 240.174,A -85,B 0,C 180,E1 -2059.238,E2 -2059.238} C_VEL
LIN {X 0,Y 573.393,Z 251.677,A -85,B 0,C 180,E1 -2060.03,E2 -2060.03} C_VEL
LIN {X 0,Y 573.287,Z 261.054,A -85,B 0,C 180,E1 -2060.83,E2 -2060.83} C_VEL
LIN {X 0,Y 573.201,Z 269.612,A -85,B 0,C 180,E1 -2061.717,E2 -2061.717} C_VEL
LIN {X 0,Y 573.138,Z 277.925,A -85,B 0,C 180,E1 -2062.78,E2 -2062.78} C_VEL
LIN {X 0,Y 573.065,Z 284.621,A -85,B 0,C 180,E1 -2063.84,E2 -2063.84} C_VEL
LIN {X 0,Y 572.962,Z 290.763,A -85,B 0,C 180,E1 -2065.075,E2 -2065.075} C_VEL
LIN {X 0,Y 573.015,Z 294.752,A -85,B 0,C 180,E1 -2066.132,E2 -2066.132} C_VEL
LIN {X 0,Y 572.959,Z 297.701,A -85,B 0,C 180,E1 -2067.188,E2 -2067.188} C_VEL
LIN {X 0,Y 572.94,Z 299.127,A -85,B 0,C 180,E1 -2067.891,E2 -2067.891} C_VEL
LIN {X 0,Y 572.941,Z 300.756,A -85,B 0,C 180,E1 -2069.297,E2 -2069.297} C_VEL
LIN {X 0,Y 572.939,Z 300.996,A -85,B 0,C 180,E1 -2070,E2 -2070} C_VEL
LIN {X 0,Y 572.94,Z 300.815,A -85,B 0,C 180,E1 -2070.703,E2 -2070.703} C_VEL
LIN {X 0,Y 572.94,Z 299.269,A -85,B 0,C 180,E1 -2072.109,E2 -2072.109} C_VEL
LIN {X 0,Y 572.96,Z 297.908,A -85,B 0,C 180,E1 -2072.812,E2 -2072.812} C_VEL
LIN {X 0,Y 573.015,Z 295.031,A -85,B 0,C 180,E1 -2073.868,E2 -2073.868} C_VEL
LIN {X 0,Y 572.963,Z 291.131,A -85,B 0,C 180,E1 -2074.926,E2 -2074.926} C_VEL
LIN {X 0,Y 573.076,Z 286.099,A -85,B 0,C 180,E1 -2075.984,E2 -2075.984} C_VEL
LIN {X 0,Y 573.083,Z 279.775,A -85,B 0,C 180,E1 -2077.044,E2 -2077.044} C_VEL
LIN {X 0,Y 573.175,Z 271.854,A -85,B 0,C 180,E1 -2078.106,E2 -2078.106} C_VEL
LIN {X 0,Y 573.287,Z 262.003,A -85,B 0,C 180,E1 -2079.17,E2 -2079.17} C_VEL
LIN {X 0,Y 573.406,Z 251.684,A -85,B 0,C 180,E1 -2080.059,E2 -2080.059} C_VEL
LIN {X 0,Y 573.485,Z 240.266,A -85,B 0,C 180,E1 -2080.847,E2 -2080.847} C_VEL
LIN {X 0,Y 573.585,Z 229.197,A -85,B 0,C 180,E1 -2081.451,E2 -2081.451} C_VEL
LIN {X 0,Y 573.726,Z 216.606,A -85,B 0,C 180,E1 -2081.97,E2 -2081.97} C_VEL
LIN {X 0,Y 573.847,Z 203.436,A -85,B 0,C 180,E1 -2082.354,E2 -2082.354} C_VEL
LIN {X 0,Y 573.346,Z 199.093,A -85,B 0,C 180,E1 -2082.457,E2 -2082.457} C_VEL
LIN {X 0,Y 572.969,Z 196.53,A -85,B 0,C 180,E1 -2082.53,E2 -2082.53} C_VEL
LIN {X 0,Y 572.969,Z 191.949,A -85,B 0,C 180,E1 -2084.927,E2 -2084.927} C_VEL
LIN {X 0,Y 572.967,Z 186.416,A -85,B 0,C 180,E1 -2087.858,E2 -2087.858} C_VEL
LIN {X 0,Y 573.015,Z 182.296,A -85,B 0,C 180,E1 -2090.085,E2 -2090.085} C_VEL
LIN {X 0,Y 573.091,Z 176.902,A -85,B 0,C 180,E1 -2093.11,E2 -2093.11} C_VEL
LIN {X 0,Y 573.095,Z 172.891,A -85,B 0,C 180,E1 -2095.418,E2 -2095.418} C_VEL
LIN {X 0,Y 573.14,Z 168.435,A -85,B 0,C 180,E1 -2098.007,E2 -2098.007} C_VEL
LIN {X 0,Y 573.154,Z 163.434,A -85,B 0,C 180,E1 -2100.998,E2 -2100.998} C_VEL
LIN {X 0,Y 573.177,Z 159.268,A -85,B 0,C 180,E1 -2103.51,E2 -2103.51} C_VEL
LIN {X 0,Y 573.181,Z 156.506,A -85,B 0,C 180,E1 -2105.19,E2 -2105.19} C_VEL
LIN {X 0,Y 573.186,Z 156.084,A -85,B 0,C 180,E1 -2106.054,E2 -2106.054} C_VEL
LIN {X 0,Y 573.218,Z 156.086,A -85,B 0,C 180,E1 -2108.704,E2 -2108.704} C_VEL
LIN {X 0,Y 573.21,Z 156.081,A -85,B 0,C 180,E1 -2111.459,E2 -2111.459} C_VEL
LIN {X 0,Y 573.235,Z 156.079,A -85,B 0,C 180,E1 -2114.334,E2 -2114.334} C_VEL
LIN {X 0,Y 573.242,Z 156.082,A -85,B 0,C 180,E1 -2117.358,E2 -2117.358} C_VEL
LIN {X 0,Y 573.238,Z 156.08,A -85,B 0,C 180,E1 -2120.392,E2 -2120.392} C_VEL
LIN {X 0,Y 573.22,Z 156.08,A -85,B 0,C 180,E1 -2123.075,E2 -2123.075} C_VEL
LIN {X 0,Y 573.249,Z 156.082,A -85,B 0,C 180,E1 -2125.67,E2 -2125.67} C_VEL
LIN {X 0,Y 573.242,Z 156.077,A -85,B 0,C 180,E1 -2128.184,E2 -2128.184} C_VEL
LIN {X 0,Y 573.266,Z 156.077,A -85,B 0,C 180,E1 -2130.634,E2 -2130.634} C_VEL
LIN {X 0,Y 573.252,Z 156.078,A -85,B 0,C 180,E1 -2133.024,E2 -2133.024} C_VEL
LIN {X 0,Y 573.275,Z 156.072,A -85,B 0,C 180,E1 -2135.366,E2 -2135.366} C_VEL
LIN {X 0,Y 573.221,Z 156.08,A -85,B 0,C 180,E1 -2138.419,E2 -2138.419} C_VEL
LIN {X 0,Y 573.27,Z 156.075,A -85,B 0,C 180,E1 -2140.731,E2 -2140.731} C_VEL
LIN {X 0,Y 573.251,Z 156.076,A -85,B 0,C 180,E1 -2143.622,E2 -2143.622} C_VEL
LIN {X 0,Y 573.274,Z 156.074,A -85,B 0,C 180,E1 -2145.807,E2 -2145.807} C_VEL
LIN {X 0,Y 573.264,Z 156.074,A -85,B 0,C 180,E1 -2148.745,E2 -2148.745} C_VEL
LIN {X 0,Y 573.238,Z 156.084,A -85,B 0,C 180,E1 -2151.54,E2 -2151.54} C_VEL
LIN {X 0,Y 573.266,Z 156.075,A -85,B 0,C 180,E1 -2154.372,E2 -2154.372} C_VEL
LIN {X 0,Y 573.302,Z 156.07,A -85,B 0,C 180,E1 -2157.189,E2 -2157.189} C_VEL
LIN {X 0,Y 573.323,Z 156.073,A -85,B 0,C 180,E1 -2160,E2 -2160} C_VEL
LIN {X 0,Y 573.304,Z 156.069,A -85,B 0,C 180,E1 -2162.811,E2 -2162.811} C_VEL
LIN {X 0,Y 573.275,Z 156.074,A -85,B 0,C 180,E1 -2165.628,E2 -2165.628} C_VEL
LIN {X 0,Y 573.235,Z 156.082,A -85,B 0,C 180,E1 -2168.46,E2 -2168.46} C_VEL
LIN {X 0,Y 573.273,Z 156.073,A -85,B 0,C 180,E1 -2171.312,E2 -2171.312} C_VEL
LIN {X 0,Y 573.283,Z 156.072,A -85,B 0,C 180,E1 -2174.424,E2 -2174.424} C_VEL
LIN {X 0,Y 573.259,Z 156.081,A -85,B 0,C 180,E1 -2177.112,E2 -2177.112} C_VEL
LIN {X 0,Y 573.239,Z 156.078,A -85,B 0,C 180,E1 -2180.077,E2 -2180.077} C_VEL
LIN {X 0,Y 573.226,Z 156.086,A -85,B 0,C 180,E1 -2182.338,E2 -2182.338} C_VEL
LIN {X 0,Y 573.246,Z 156.079,A -85,B 0,C 180,E1 -2185.411,E2 -2185.411} C_VEL
LIN {X 0,Y 573.235,Z 156.078,A -85,B 0,C 180,E1 -2188.565,E2 -2188.565} C_VEL
LIN {X 0,Y 573.228,Z 156.085,A -85,B 0,C 180,E1 -2190.993,E2 -2190.993} C_VEL
LIN {X 0,Y 573.264,Z 156.074,A -85,B 0,C 180,E1 -2193.524,E2 -2193.524} C_VEL
LIN {X 0,Y 573.186,Z 156.09,A -85,B 0,C 180,E1 -2196.054,E2 -2196.054} C_VEL
LIN {X 0,Y 573.228,Z 156.078,A -85,B 0,C 180,E1 -2198.703,E2 -2198.703} C_VEL
LIN {X 0,Y 573.229,Z 156.08,A -85,B 0,C 180,E1 -2201.593,E2 -2201.593} C_VEL
LIN {X 0,Y 573.226,Z 156.083,A -85,B 0,C 180,E1 -2204.335,E2 -2204.335} C_VEL
LIN {X 0,Y 573.242,Z 156.077,A -85,B 0,C 180,E1 -2207.359,E2 -2207.359} C_VEL
LIN {X 0,Y 573.232,Z 156.079,A -85,B 0,C 180,E1 -2210.392,E2 -2210.392} C_VEL
LIN {X 0,Y 573.236,Z 156.084,A -85,B 0,C 180,E1 -2213.569,E2 -2213.569} C_VEL
LIN {X 0,Y 573.581,Z 159.169,A -85,B 0,C 180,E1 -2214.838,E2 -2214.838} C_VEL
LIN {X 0,Y 573.475,Z 166.831,A -85,B 0,C 180,E1 -2217.737,E2 -2217.737} C_VEL
LIN {X 0,Y 573.456,Z 174.752,A -85,B 0,C 180,E1 -2220.645,E2 -2220.645} C_VEL
LIN {X 0,Y 573.314,Z 183.656,A -85,B 0,C 180,E1 -2223.813,E2 -2223.813} C_VEL
LIN {X 0,Y 573.248,Z 191.449,A -85,B 0,C 180,E1 -2226.519,E2 -2226.519} C_VEL
LIN {X 0,Y 573.176,Z 199.239,A -85,B 0,C 180,E1 -2229.171,E2 -2229.171} C_VEL
LIN {X 0,Y 573.133,Z 207.03,A -85,B 0,C 180,E1 -2231.778,E2 -2231.778} C_VEL
LIN {X 0,Y 573.102,Z 214.822,A -85,B 0,C 180,E1 -2234.348,E2 -2234.348} C_VEL
LIN {X 0,Y 573.063,Z 222.613,A -85,B 0,C 180,E1 -2236.886,E2 -2236.886} C_VEL
LIN {X 0,Y 573.032,Z 224.491,A -85,B 0,C 180,E1 -2237.494,E2 -2237.494} C_VEL
LIN {X 0,Y 573.87,Z 230.365,A -85,B 0,C 180,E1 -2237.624,E2 -2237.624} C_VEL
LIN {X 0,Y 573.764,Z 242.492,A -85,B 0,C 180,E1 -2237.936,E2 -2237.936} C_VEL
LIN {X 0,Y 573.625,Z 255.391,A -85,B 0,C 180,E1 -2238.421,E2 -2238.421} C_VEL
LIN {X 0,Y 573.52,Z 266.666,A -85,B 0,C 180,E1 -2238.987,E2 -2238.987} C_VEL
LIN {X 0,Y 573.435,Z 277.476,A -85,B 0,C 180,E1 -2239.674,E2 -2239.674} C_VEL
LIN {X 0,Y 573.307,Z 287.645,A -85,B 0,C 180,E1 -2240.474,E2 -2240.474} C_VEL
LIN {X 0,Y 573.215,Z 296.786,A -85,B 0,C 180,E1 -2241.362,E2 -2241.362} C_VEL
LIN {X 0,Y 573.142,Z 305.689,A -85,B 0,C 180,E1 -2242.425,E2 -2242.425} C_VEL
LIN {X 0,Y 573.051,Z 312.405,A -85,B 0,C 180,E1 -2243.415,E2 -2243.415} C_VEL
LIN {X 0,Y 573.07,Z 317.68,A -85,B 0,C 180,E1 -2244.369,E2 -2244.369} C_VEL
LIN {X 0,Y 573.028,Z 322.371,A -85,B 0,C 180,E1 -2245.427,E2 -2245.427} C_VEL
LIN {X 0,Y 573.022,Z 325.956,A -85,B 0,C 180,E1 -2246.484,E2 -2246.484} C_VEL
LIN {X 0,Y 572.959,Z 327.808,A -85,B 0,C 180,E1 -2247.188,E2 -2247.188} C_VEL
LIN {X 0,Y 572.94,Z 329.2,A -85,B 0,C 180,E1 -2247.891,E2 -2247.891} C_VEL
LIN {X 0,Y 572.94,Z 330.784,A -85,B 0,C 180,E1 -2249.297,E2 -2249.297} C_VEL
LIN {X 0,Y 572.938,Z 331,A -85,B 0,C 180,E1 -2250,E2 -2250} C_VEL
LIN {X 0,Y 572.946,Z 330.185,A -85,B 0,C 180,E1 -2251.406,E2 -2251.406} C_VEL
LIN {X 0,Y 572.94,Z 329.202,A -85,B 0,C 180,E1 -2252.109,E2 -2252.109} C_VEL
LIN {X 0,Y 572.959,Z 327.81,A -85,B 0,C 180,E1 -2252.812,E2 -2252.812} C_VEL
LIN {X 0,Y 573.014,Z 324.897,A -85,B 0,C 180,E1 -2253.868,E2 -2253.868} C_VEL
LIN {X 0,Y 572.963,Z 320.95,A -85,B 0,C 180,E1 -2254.925,E2 -2254.925} C_VEL
LIN {X 0,Y 573.065,Z 314.879,A -85,B 0,C 180,E1 -2256.16,E2 -2256.16} C_VEL
LIN {X 0,Y 573.119,Z 308.238,A -85,B 0,C 180,E1 -2257.221,E2 -2257.221} C_VEL
LIN {X 0,Y 573.201,Z 299.991,A -85,B 0,C 180,E1 -2258.283,E2 -2258.283} C_VEL
LIN {X 0,Y 573.287,Z 291.54,A -85,B 0,C 180,E1 -2259.17,E2 -2259.17} C_VEL
LIN {X 0,Y 573.412,Z 281.097,A -85,B 0,C 180,E1 -2260.058,E2 -2260.058} C_VEL
LIN {X 0,Y 573.469,Z 270.9,A -85,B 0,C 180,E1 -2260.763,E2 -2260.763} C_VEL
LIN {X 0,Y 573.602,Z 258.854,A -85,B 0,C 180,E1 -2261.422,E2 -2261.422} C_VEL
LIN {X 0,Y 573.733,Z 246.478,A -85,B 0,C 180,E1 -2261.929,E2 -2261.929} C_VEL
LIN {X 0,Y 573.864,Z 233.445,A -85,B 0,C 180,E1 -2262.308,E2 -2262.308} C_VEL
LIN {X 0,Y 573.669,Z 228.664,A -85,B 0,C 180,E1 -2262.413,E2 -2262.413} C_VEL
LIN {X 0,Y 573.032,Z 224.492,A -85,B 0,C 180,E1 -2262.506,E2 -2262.506} C_VEL
LIN {X 0,Y 573.082,Z 215.936,A -85,B 0,C 180,E1 -2265.287,E2 -2265.287} C_VEL
LIN {X 0,Y 573.14,Z 208.144,A -85,B 0,C 180,E1 -2267.852,E2 -2267.852} C_VEL
LIN {X 0,Y 573.195,Z 200.353,A -85,B 0,C 180,E1 -2270.453,E2 -2270.453} C_VEL
LIN {X 0,Y 573.224,Z 192.44,A -85,B 0,C 180,E1 -2273.141,E2 -2273.141} C_VEL
LIN {X 0,Y 573.29,Z 184.77,A -85,B 0,C 180,E1 -2275.798,E2 -2275.798} C_VEL
LIN {X 0,Y 573.363,Z 176.979,A -85,B 0,C 180,E1 -2278.557,E2 -2278.557} C_VEL
LIN {X 0,Y 573.458,Z 170.301,A -85,B 0,C 180,E1 -2280.979,E2 -2280.979} C_VEL
LIN {X 0,Y 573.536,Z 163.357,A -85,B 0,C 180,E1 -2283.565,E2 -2283.565} C_VEL
LIN {X 0,Y 573.534,Z 158.099,A -85,B 0,C 180,E1 -2285.579,E2 -2285.579} C_VEL
LIN {X 0,Y 573.235,Z 156.084,A -85,B 0,C 180,E1 -2286.431,E2 -2286.431} C_VEL
LIN {X 0,Y 573.231,Z 156.079,A -85,B 0,C 180,E1 -2289.608,E2 -2289.608} C_VEL
LIN {X 0,Y 573.24,Z 156.078,A -85,B 0,C 180,E1 -2292.641,E2 -2292.641} C_VEL
LIN {X 0,Y 573.224,Z 156.083,A -85,B 0,C 180,E1 -2295.665,E2 -2295.665} C_VEL
LIN {X 0,Y 573.227,Z 156.082,A -85,B 0,C 180,E1 -2298.543,E2 -2298.543} C_VEL
LIN {X 0,Y 573.23,Z 156.078,A -85,B 0,C 180,E1 -2301.297,E2 -2301.297} C_VEL
LIN {X 0,Y 573.184,Z 156.091,A -85,B 0,C 180,E1 -2304.022,E2 -2304.022} C_VEL
LIN {X 0,Y 573.268,Z 156.074,A -85,B 0,C 180,E1 -2306.518,E2 -2306.518} C_VEL
LIN {X 0,Y 573.234,Z 156.084,A -85,B 0,C 180,E1 -2309.116,E2 -2309.116} C_VEL
LIN {X 0,Y 573.235,Z 156.079,A -85,B 0,C 180,E1 -2311.435,E2 -2311.435} C_VEL
LIN {X 0,Y 573.262,Z 156.076,A -85,B 0,C 180,E1 -2313.81,E2 -2313.81} C_VEL
